   VAR
      s_UDT_MessageArray { ExternalAccessible := 'False'; ExternalVisible := 'False'; ExternalWritable := 'False'; S7_SetPoint := 'False'} : "UDT_MessageV2";   // Message array byte
      s_UDT_MessageHeader { ExternalAccessible := 'False'; ExternalVisible := 'False'; ExternalWritable := 'False'; S7_SetPoint := 'False'} : "UDT_MFCSortMessageHeader";   // Message header
      s_F_TRIG_SendAllStatuses {InstructionName := 'F_TRIG'; LibVersion := '1.0'; ExternalAccessible := 'False'; ExternalVisible := 'False'; ExternalWritable := 'False'; S7_SetPoint := 'False'} : F_TRIG;   // Falling edge trigger from signal send all statuses
      ss_MessageBody { ExternalAccessible := 'False'; ExternalVisible := 'False'; ExternalWritable := 'False'} : Struct   // Message body
         MsgID { ExternalAccessible := 'False'; ExternalVisible := 'False'; ExternalWritable := 'False'} : Word;   // Message ID
         MsgLength { ExternalAccessible := 'False'; ExternalVisible := 'False'; ExternalWritable := 'False'} : Word;   // Message length
         SystemStatus { ExternalAccessible := 'False'; ExternalVisible := 'False'; ExternalWritable := 'False'} : Byte;   // System status
         SystemMode { ExternalAccessible := 'False'; ExternalVisible := 'False'; ExternalWritable := 'False'} : Word;   // System mode
         Eom { ExternalAccessible := 'False'; ExternalVisible := 'False'; ExternalWritable := 'False'} : Byte;   // End of message
      END_STRUCT;
      ss_Status { ExternalAccessible := 'False'; ExternalVisible := 'False'; ExternalWritable := 'False'} : Struct   // Status structure
         FIFOStatus { ExternalAccessible := 'False'; ExternalVisible := 'False'; ExternalWritable := 'False'} : "UDT_FifoStatus";
         FIFOError { ExternalAccessible := 'False'; ExternalVisible := 'False'; ExternalWritable := 'False'; S7_SetPoint := 'True'} : Bool;   //  FIFO error
         FIFOWarning { ExternalAccessible := 'False'; ExternalVisible := 'False'; ExternalWritable := 'False'; S7_SetPoint := 'True'} : Bool;   // FIFO warning
         InvalidMessageArraySize { ExternalAccessible := 'False'; ExternalVisible := 'False'; ExternalWritable := 'False'} : Bool;   // Message array is too short for message
         InvalidTimeInterval { ExternalAccessible := 'False'; ExternalVisible := 'False'; ExternalWritable := 'False'} : Bool;   // Heartbeat time interval lower than zero
      END_STRUCT;
      sdi_SerializePosition { ExternalAccessible := 'False'; ExternalVisible := 'False'; ExternalWritable := 'False'} : DInt;   // Position in array where serialize finished writing data +1
      si_MaximumMessageLength { ExternalAccessible := 'False'; ExternalVisible := 'False'; ExternalWritable := 'False'} : Int;   // Maximum number of elements in message array
      si_SerializeStatus { ExternalAccessible := 'False'; ExternalVisible := 'False'; ExternalWritable := 'False'} : Int;   // Function serialize status
      si_SystemStatus { ExternalAccessible := 'False'; ExternalVisible := 'False'; ExternalWritable := 'False'} : Int := 0;   // 0 - System stopped, 1 - System running
      sw_SystemMode { ExternalAccessible := 'False'; ExternalVisible := 'False'; ExternalWritable := 'False'} : Word := 0;   // Bit value according to the documentation
      si_Old_SystemStatus { ExternalAccessible := 'False'; ExternalVisible := 'False'; ExternalWritable := 'False'} : Int := 0;   // Data from previous PLC cycle: 0 - System stopped, 1 - System running
      sw_Old_SystemMode { ExternalAccessible := 'False'; ExternalVisible := 'False'; ExternalWritable := 'False'} : Word := 0;   // Bit value according to the documentation
      sx_NewData { ExternalAccessible := 'False'; ExternalVisible := 'False'; ExternalWritable := 'False'} : Bool;   // True - send a message to the MFC
   END_VAR

   VAR CONSTANT
      ci_MessageLength : Word := 16#0006;   // 10#0006 = 16#0006 - Message length
      ci_Som : Byte := 16#FD;   // Start of message
      ci_Eom : Byte := 16#FE;   // End of message
      ci_MsgID : Word := 16#00CC;   // 10#0204 = 16#00CC - Message ID
      ci_MsgLength : Word := 16#0002;   // 10#0002 = 16#0002 - Message length
   END_VAR


BEGIN
	(*
	----------------------------------------------------------------------------------------
	|                                                                                      |
	|  Copyright  2023             FORTNA Europe BV                                        |
	|  All Rights Reserved         Netherlands                                             |
	|                                                                                      |
	----------------------------------------------------------------------------------------
	Version history:
	Date        | Version   | Author       | Remark
	----------------------------------------------------------------------------------------
	25/04/2023  | 1.0       | S. Nikodem   | Release TIA 17 | DHL Munich 2023
	13/09/2023  | 1.1       | S. Nikodem   | Change type of variable System mode to word
	20/10/2023  | 1.2       | S. Nikodem   | Added "ix_SendAllStatuses" input and update for Serialize structure
	13/03/2023  | 1.3       | S. Nieswiec  | Updated for new Baseline
	02/05/2024  | 1.4       | J.Majer      | Datatype conversions changed from automatic to explicit, to accomodate IEC 61131-3 standard

	*)

	REGION 1 – FIFO header status update

	    // Mode 'S' - FIFO register status update.
	    "FC_Fifo"(ic_Mode := 'S',
	              qUDT_Status => #ss_Status.FIFOStatus,
	              qx_Error => #ss_Status.FIFOError,
	              qx_Warning => #ss_Status.FIFOWarning,
	              iqv_Data := #s_UDT_MessageArray,
	              iqUDT_FifoHeader := #iq_UDT_FifoHeader,
	              iqv_DataBuffer := #iqa_FifoData);

	END_REGION

	REGION 2 – Data preparation

	    // Prepare trigger
	    #s_F_TRIG_SendAllStatuses(CLK := #ix_SendAllStatuses);

	    // Data preparation
	    //  1 - System stopped, 2 - System running
	    #si_SystemStatus := #ii_SystemStatus;
	    // Bit value according to the documentation
	    #sw_SystemMode := #iw_SystemMode;

	    //Check if the data from the previous PLC cycle differs, if so, send a message to the MFC.
	    #sx_NewData := (#si_Old_SystemStatus <> #si_SystemStatus) OR (#sw_Old_SystemMode <> #sw_SystemMode) OR #s_F_TRIG_SendAllStatuses.Q;

	    // Copy data
	    #si_Old_SystemStatus := #si_SystemStatus;
	    #sw_Old_SystemMode := #sw_SystemMode;

	END_REGION

	REGION 3 – Message array size validation

	    // Get size of the array.
	    #si_MaximumMessageLength := "FC_GetNrOfArrayEl"(#s_UDT_MessageArray.Bytes);

	    // Message array size validation.
	    #ss_Status.InvalidMessageArraySize := WORD_TO_INT(#ci_MessageLength) > #si_MaximumMessageLength;

	END_REGION

	REGION 4 – Message preparation

	    // FIFO full check.
	    IF NOT #iq_UDT_FifoHeader.Status.Full
	    THEN
	        // Errors and send pulse check.
	        IF NOT #ss_Status.FIFOError
	            AND NOT #ss_Status.InvalidMessageArraySize
	            AND #sx_NewData
	        THEN

	            REGION 4.1 – Header preparation

	                // Check sequence number. If it is equal or greater than 255 reset it to 1.
	                IF #iqi_MessageSequenceNumber <= 255
	                THEN
	                    #iqi_MessageSequenceNumber += 1;
	                ELSE
	                    #iqi_MessageSequenceNumber := 1;
	                END_IF;

	                // Write parts of the header into structure.
	                #s_UDT_MessageHeader.SOM := #ci_Som;
	                #s_UDT_MessageHeader.SourceNode := INT_TO_BYTE(#ii_SourceNode);
	                #s_UDT_MessageHeader.DestinationNode := INT_TO_BYTE(#ii_DestinationNode);
	                #s_UDT_MessageHeader.SeqNumber := INT_TO_BYTE(#iqi_MessageSequenceNumber);
	                #s_UDT_MessageHeader.DataLength := #ci_MessageLength;
	                #s_UDT_MessageHeader.NumMsg := 1;

	                // Write parts of the body into structure.
	                #ss_MessageBody.MsgID := #ci_MsgID;
	                #ss_MessageBody.MsgLength := #ci_MsgLength;
	                #ss_MessageBody.SystemStatus := INT_TO_BYTE(#si_SystemStatus);
	                #ss_MessageBody.SystemMode := #sw_SystemMode;
	                #ss_MessageBody.Eom := #ci_Eom;

	            END_REGION

	            REGION 4.2 – Convert message into array of bytes

	                // Initialize the header serialize position and convert header structure into array of bytes.
	                #sdi_SerializePosition := 0;
	                #si_SerializeStatus := Serialize(SRC_VARIABLE := #s_UDT_MessageHeader,
	                                                 DEST_ARRAY => #s_UDT_MessageArray.Bytes,
	                                                 POS := #sdi_SerializePosition);

	                #si_SerializeStatus := Serialize(SRC_VARIABLE := #ss_MessageBody.MsgID,
	                                                 DEST_ARRAY => #s_UDT_MessageArray.Bytes,
	                                                 POS := #sdi_SerializePosition);

	                #si_SerializeStatus := Serialize(SRC_VARIABLE := #ss_MessageBody.MsgLength,
	                                                 DEST_ARRAY => #s_UDT_MessageArray.Bytes,
	                                                 POS := #sdi_SerializePosition);

	                #si_SerializeStatus := Serialize(SRC_VARIABLE := #ss_MessageBody.SystemStatus,
	                                                 DEST_ARRAY => #s_UDT_MessageArray.Bytes,
	                                                 POS := #sdi_SerializePosition);

	                #si_SerializeStatus := Serialize(SRC_VARIABLE := #ss_MessageBody.SystemMode,
	                                                 DEST_ARRAY => #s_UDT_MessageArray.Bytes,
	                                                 POS := #sdi_SerializePosition);

	                #si_SerializeStatus := Serialize(SRC_VARIABLE := #ss_MessageBody.Eom,
	                                                 DEST_ARRAY => #s_UDT_MessageArray.Bytes,
	                                                 POS := #sdi_SerializePosition);

	            END_REGION

	            REGION 4.3 – Write message into the FIFO buffer

	                // Mode 'W' - Write FIFO record.
	                "FC_Fifo"(ic_Mode := 'W',
	                          qUDT_Status => #ss_Status.FIFOStatus,
	                          qx_Error => #ss_Status.FIFOError,
	                          qx_Warning => #ss_Status.FIFOWarning,
	                          iqv_Data := #s_UDT_MessageArray,
	                          iqUDT_FifoHeader := #iq_UDT_FifoHeader,
	                          iqv_DataBuffer := #iqa_FifoData);

	            END_REGION

	        END_IF;
	    ELSE
	        // If FIFO is full set FIFO main and FIFO full errors.
	        #ss_Status.FIFOError := TRUE;
	        #ss_Status.FIFOStatus.FifoFull := TRUE;
	    END_IF;

	END_REGION

	REGION 5 - Status

	    // Parametrization collective error output.
	    #qx_Error :=
	    #ss_Status.FIFOError
	    OR #ss_Status.InvalidTimeInterval
	    OR #ss_Status.InvalidMessageArraySize;

	    // Parametrization collective warning output.
	    #qx_Warning := #ss_Status.FIFOWarning;

	END_REGION
END_FUNCTION_BLOCK

FUNCTION_BLOCK "FB_MFC_Sort_COY_Result"
{ S7_Optimized_Access := 'TRUE' }
VERSION : 0.1
// ATTRIBUTES
// AUTO_NUMBER = True
// BLOCK_NUMBER = 117
// END_ATTRIBUTES
   VAR_INPUT
      ii_GINRangeStart { ExternalAccessible := 'False'; ExternalVisible := 'False'; ExternalWritable := 'False'} : Int := 0;   // GIN range start value
      ii_GINRangeEnd { ExternalAccessible := 'False'; ExternalVisible := 'False'; ExternalWritable := 'False'} : Int := 0;   // GIN range end value
      is_ObjectID { ExternalAccessible := 'False'; ExternalVisible := 'False'; ExternalWritable := 'False'} : String[10];   // Recived parcel identifier
      ii_SourceNode { ExternalAccessible := 'False'; ExternalVisible := 'False'; ExternalWritable := 'False'} : Int;   // ID Source Node
      ii_DestinationNode { ExternalAccessible := 'False'; ExternalVisible := 'False'; ExternalWritable := 'False'} : Int;   // ID Destination Node
   END_VAR

   VAR_OUTPUT
      qx_Error { ExternalAccessible := 'False'; ExternalVisible := 'False'; ExternalWritable := 'False'} : Bool;   // TRUE when collective block error occurred
      qx_Warning { ExternalAccessible := 'False'; ExternalVisible := 'False'; ExternalWritable := 'False'} : Bool;   // TRUE when collective block warning occurred
   END_VAR

   VAR_IN_OUT
      iq_UDT_FifoHeader : "UDT_FifoHeader";   // FIFO header
      iqa_FifoData : Array[*] of "UDT_MessageV2";   // FIFO data buffer
      iqi_MessageSequenceNumber { ExternalAccessible := 'False'; ExternalVisible := 'False'; ExternalWritable := 'False'} : Int;   // Message number
   END_VAR

   VAR
      ss_FB_HeartbeatPulse { ExternalAccessible := 'False'; ExternalVisible := 'False'; ExternalWritable := 'False'; S7_SetPoint := 'False'} : "FB_Pulse";   // Heartbeat send pulse generator
      s_UDT_MessageArray { ExternalAccessible := 'False'; ExternalVisible := 'False'; ExternalWritable := 'False'; S7_SetPoint := 'False'} : "UDT_MessageV2";   // Message array byte
      s_UDT_MessageHeader { ExternalAccessible := 'False'; ExternalVisible := 'False'; ExternalWritable := 'False'; S7_SetPoint := 'False'} : "UDT_MFCSortMessageHeader";   // Message header
      ss_MessageBody { ExternalAccessible := 'False'; ExternalVisible := 'False'; ExternalWritable := 'False'} : Struct   // Message body
         MsgID { ExternalAccessible := 'False'; ExternalVisible := 'False'; ExternalWritable := 'False'} : Word;   // Message ID
         MsgLength { ExternalAccessible := 'False'; ExternalVisible := 'False'; ExternalWritable := 'False'} : Word;   // Message length
         VID { ExternalAccessible := 'False'; ExternalVisible := 'False'; ExternalWritable := 'False'} : Array[1..16] of Byte;   // Virtual Item Identifier
         PieceID { ExternalAccessible := 'False'; ExternalVisible := 'False'; ExternalWritable := 'False'} : Array[1..40] of Byte;   // Piece ID
         Group { ExternalAccessible := 'False'; ExternalVisible := 'False'; ExternalWritable := 'False'} : Byte;   // Group
         Level { ExternalAccessible := 'False'; ExternalVisible := 'False'; ExternalWritable := 'False'} : Byte;   // Level
         Result { ExternalAccessible := 'False'; ExternalVisible := 'False'; ExternalWritable := 'False'} : Byte;   // Result
         Eom { ExternalAccessible := 'False'; ExternalVisible := 'False'; ExternalWritable := 'False'} : Byte;   // End of message
      END_STRUCT;
      ss_MessageData { ExternalAccessible := 'False'; ExternalVisible := 'False'; ExternalWritable := 'False'} : Struct   // Message data
         VID { ExternalAccessible := 'False'; ExternalVisible := 'False'; ExternalWritable := 'False'} : Array[1..16] of Byte;   // Virtual Item Identifier
         PieceID { ExternalAccessible := 'False'; ExternalVisible := 'False'; ExternalWritable := 'False'} : Array[1..40] of Byte;   // Piece ID
         Group { ExternalAccessible := 'False'; ExternalVisible := 'False'; ExternalWritable := 'False'} : String[1];   // Group
         Level { ExternalAccessible := 'False'; ExternalVisible := 'False'; ExternalWritable := 'False'} : String[1];   // Level
         Result { ExternalAccessible := 'False'; ExternalVisible := 'False'; ExternalWritable := 'False'} : String[1];   // Result
      END_STRUCT;
      ss_Status { ExternalAccessible := 'False'; ExternalVisible := 'False'; ExternalWritable := 'False'} : Struct   // Status structure
         FIFOStatus { ExternalAccessible := 'False'; ExternalVisible := 'False'; ExternalWritable := 'False'} : "UDT_FifoStatus";
         FIFOError { ExternalAccessible := 'False'; ExternalVisible := 'False'; ExternalWritable := 'False'; S7_SetPoint := 'True'} : Bool;   //  FIFO error
         FIFOWarning { ExternalAccessible := 'False'; ExternalVisible := 'False'; ExternalWritable := 'False'; S7_SetPoint := 'True'} : Bool;   // FIFO warning
         InvalidMessageArraySize { ExternalAccessible := 'False'; ExternalVisible := 'False'; ExternalWritable := 'False'} : Bool;   // Message array is too short for message
         InvalidTimeInterval { ExternalAccessible := 'False'; ExternalVisible := 'False'; ExternalWritable := 'False'} : Bool;   // Heartbeat time interval lower than zero
      END_STRUCT;
      sS_Old_Object_ID { ExternalAccessible := 'False'; ExternalVisible := 'False'; ExternalWritable := 'False'} : String[10];   // Value from previous PLC cycle
      sdi_SerializePosition { ExternalAccessible := 'False'; ExternalVisible := 'False'; ExternalWritable := 'False'} : DInt;   // Position in array where serialize finished writing data +1
      si_MaximumMessageLength { ExternalAccessible := 'False'; ExternalVisible := 'False'; ExternalWritable := 'False'} : Int;   // Maximum number of elements in message array
      si_SerializeStatus { ExternalAccessible := 'False'; ExternalVisible := 'False'; ExternalWritable := 'False'} : Int;   // Function serialize status
      sx_NewData { ExternalAccessible := 'False'; ExternalVisible := 'False'; ExternalWritable := 'False'} : Bool;   // True - send a message to the MFC
   END_VAR

   VAR_TEMP
      ti_Loop_GIN : Int;   // Loop counter for DB_GIN
      ti_Loop : Int;   // Loop counter
   END_VAR

   VAR CONSTANT
      ci_MessageLength : Word := 16#003F;   // 10#0063 = 16#003F - Message length
      ci_MsgID : Word := 16#0137;   // 10#0311 = 16#0137 - Message ID
      ci_MsgLength : Word := 16#003B;   // 10#0059 = 16#003B - Message length
      ci_Som : Byte := 16#FD;   // Start of message
      ci_Eom : Byte := 16#FE;   // End of message
   END_VAR


BEGIN
	(*
	----------------------------------------------------------------------------------------
	|                                                                                      |
	|  Copyright  2023             FORTNA Europe BV                                        |
	|  All Rights Reserved         Netherlands                                             |
	|                                                                                      |
	----------------------------------------------------------------------------------------
	Version history:
	Date        | Version   | Author       | Remark
	----------------------------------------------------------------------------------------
	24/04/2023  | 1.0       | S. Nikodem   | Release TIA 17 | DHL Munich 2023
	03/10/2023  | 1.1       | S. Nikodem   | Update
	13/03/2023  | 1.2       | S. Nieswiec  | Updated for new Baseline
	02/05/2024  | 1.3       | J.Majer      | Datatype conversions changed from automatic to explicit, to accomodate IEC 61131-3 standard
	*)

	REGION 1 – FIFO header status update

	    // Mode 'S' - FIFO register status update.
	    "FC_Fifo"(ic_Mode := 'S',
	              qUDT_Status => #ss_Status.FIFOStatus,
	              qx_Error => #ss_Status.FIFOError,
	              qx_Warning => #ss_Status.FIFOWarning,
	              iqv_Data := #s_UDT_MessageArray,
	              iqUDT_FifoHeader := #iq_UDT_FifoHeader,
	              iqv_DataBuffer := #iqa_FifoData);

	END_REGION

	REGION 2 – Data preparation

	    //Generation message when is new parcel
	    #sx_NewData := (#is_ObjectID <> #sS_Old_Object_ID) AND NOT (#is_ObjectID = '');
	    // Save last value
	    #sS_Old_Object_ID := #is_ObjectID;

	    IF #sx_NewData THEN

	        FOR #ti_Loop_GIN := #ii_GINRangeStart TO #ii_GINRangeEnd DO

	            IF "DB_GIN".GIN[#ti_Loop_GIN].DHL.ObjectID = #is_ObjectID THEN

	                //VID
	                FOR #ti_Loop := 1 TO 16 DO

	                    #ss_MessageData.VID[#ti_Loop] := CHAR_TO_BYTE("DB_GIN".GIN[#ti_Loop_GIN].DHL.VID[#ti_Loop]);

	                END_FOR;

	                //Piece ID
	                FOR #ti_Loop := 1 TO 40 DO

	                    #ss_MessageData.PieceID[#ti_Loop] := CHAR_TO_BYTE("DB_GIN".GIN[#ti_Loop_GIN].DHL.PieceID[#ti_Loop]);

	                END_FOR;

	                //Group
	                #ss_MessageData.Group := "DB_GIN".GIN[#ti_Loop_GIN].DHL.Xray.Group;

	                //Level
	                #ss_MessageData.Level := "DB_GIN".GIN[#ti_Loop_GIN].DHL.Xray.Level;

	                //Result
	                #ss_MessageData.Result := "DB_GIN".GIN[#ti_Loop_GIN].DHL.Xray.Result;

	            END_IF;

	        END_FOR;

	    END_IF;

	END_REGION

	REGION 3 – Message array size validation

	    // Get size of the array.
	    #si_MaximumMessageLength := "FC_GetNrOfArrayEl"(#s_UDT_MessageArray.Bytes);

	    // Message array size validation.
	    #ss_Status.InvalidMessageArraySize := WORD_TO_INT(#ci_MessageLength) > #si_MaximumMessageLength;

	END_REGION


	REGION 4 – Message preparation

	    // FIFO full check.
	    IF NOT #iq_UDT_FifoHeader.Status.Full
	    THEN
	        // Errors and send pulse check.
	        IF NOT #ss_Status.FIFOError
	            AND NOT #ss_Status.InvalidMessageArraySize
	            AND #sx_NewData
	        THEN

	            REGION 4.1 – Header preparation

	                // Check sequence number. If it is equal or greater than 255 reset it to 1.
	                IF #iqi_MessageSequenceNumber <= 255
	                THEN
	                    #iqi_MessageSequenceNumber += 1;
	                ELSE
	                    #iqi_MessageSequenceNumber := 1;
	                END_IF;

	                // Write parts of the header into structure.
	                #s_UDT_MessageHeader.SOM := #ci_Som;
	                #s_UDT_MessageHeader.SourceNode := INT_TO_BYTE(#ii_SourceNode);
	                #s_UDT_MessageHeader.DestinationNode := INT_TO_BYTE(#ii_DestinationNode);
	                #s_UDT_MessageHeader.SeqNumber := INT_TO_BYTE(#iqi_MessageSequenceNumber);
	                #s_UDT_MessageHeader.DataLength := #ci_MessageLength;
	                #s_UDT_MessageHeader.NumMsg := 1;

	                // Write parts of the body into structure.
	                #ss_MessageBody.MsgID := #ci_MsgID;
	                #ss_MessageBody.MsgLength := #ci_MsgLength;
	                #ss_MessageBody.VID := #ss_MessageData.VID;
	                #ss_MessageBody.PieceID := #ss_MessageData.PieceID;
	                #ss_MessageBody.Group := CHAR_TO_BYTE(STRING_TO_CHAR(#ss_MessageData.Group));
	                #ss_MessageBody.Level := CHAR_TO_BYTE(STRING_TO_CHAR(#ss_MessageData.Level));
	                #ss_MessageBody.Result := CHAR_TO_BYTE(STRING_TO_CHAR(#ss_MessageData.Result));
	                #ss_MessageBody.Eom := #ci_Eom;

	            END_REGION

	            REGION 4.2 – Convert message into array of bytes

	                // Initialize the header serialize position and convert header structure into array of bytes.
	                #sdi_SerializePosition := 0;
	                #si_SerializeStatus := Serialize(SRC_VARIABLE := #s_UDT_MessageHeader,
	                                                 DEST_ARRAY => #s_UDT_MessageArray.Bytes,
	                                                 POS := #sdi_SerializePosition);

	                // Initialize the body serialize position and convert header structure into array of bytes
	                #si_SerializeStatus := Serialize(SRC_VARIABLE := #ss_MessageBody,
	                                                 DEST_ARRAY => #s_UDT_MessageArray.Bytes,
	                                                 POS := #sdi_SerializePosition);

	            END_REGION

	            REGION 4.3 – Write message into the FIFO buffer

	                // Mode 'W' - Write FIFO record.
	                "FC_Fifo"(ic_Mode := 'W',
	                          qUDT_Status => #ss_Status.FIFOStatus,
	                          qx_Error => #ss_Status.FIFOError,
	                          qx_Warning => #ss_Status.FIFOWarning,
	                          iqv_Data := #s_UDT_MessageArray,
	                          iqUDT_FifoHeader := #iq_UDT_FifoHeader,
	                          iqv_DataBuffer := #iqa_FifoData);

	            END_REGION

	        END_IF;
	    ELSE
	        // If FIFO is full set FIFO main and FIFO full errors.
	        #ss_Status.FIFOError := TRUE;
	        #ss_Status.FIFOStatus.FifoFull := TRUE;
	    END_IF;

	END_REGION

	REGION 5 - Status

	    // Parametrization collective error output.
	    #qx_Error :=
	    #ss_Status.FIFOError
	    OR #ss_Status.InvalidTimeInterval
	    OR #ss_Status.InvalidMessageArraySize;

	    // Parametrization collective warning output.
	    #qx_Warning := #ss_Status.FIFOWarning;

	END_REGION
END_FUNCTION_BLOCK

FUNCTION_BLOCK "FB_MFC_Sort_COY_RegInfo"
{ S7_Optimized_Access := 'TRUE' }
VERSION : 0.1
// ATTRIBUTES
// AUTO_NUMBER = True
// BLOCK_NUMBER = 116
// END_ATTRIBUTES
   VAR_INPUT
      is_ObjectID { ExternalAccessible := 'False'; ExternalVisible := 'False'; ExternalWritable := 'False'} : String[10];   // Parcel identifier
      ii_XrayLocation { ExternalAccessible := 'False'; ExternalVisible := 'False'; ExternalWritable := 'False'} : Int;   // X-ray location
      ii_SourceNode { ExternalAccessible := 'False'; ExternalVisible := 'False'; ExternalWritable := 'False'} : Int;   // ID Source Node
      ii_DestinationNode { ExternalAccessible := 'False'; ExternalVisible := 'False'; ExternalWritable := 'False'} : Int;   // ID Destination Node
   END_VAR

   VAR_OUTPUT
      qx_Error { ExternalAccessible := 'False'; ExternalVisible := 'False'; ExternalWritable := 'False'} : Bool;   // TRUE when collective block error occurred
      qx_Warning { ExternalAccessible := 'False'; ExternalVisible := 'False'; ExternalWritable := 'False'} : Bool;   // TRUE when collective block warning occurred
   END_VAR

   VAR_IN_OUT
      iq_UDT_FifoHeader : "UDT_FifoHeader";   // FIFO header
      iqa_FifoData : Array[*] of "UDT_MessageV2";   // FIFO data buffer
      iqi_MessageSequenceNumber { ExternalAccessible := 'False'; ExternalVisible := 'False'; ExternalWritable := 'False'} : Int;   // Message number
   END_VAR

   VAR
      ss_FB_HeartbeatPulse { ExternalAccessible := 'False'; ExternalVisible := 'False'; ExternalWritable := 'False'; S7_SetPoint := 'False'} : "FB_Pulse";   // Heartbeat send pulse generator
      s_UDT_MessageArray { ExternalAccessible := 'False'; ExternalVisible := 'False'; ExternalWritable := 'False'; S7_SetPoint := 'False'} : "UDT_MessageV2";   // Message array byte
      s_UDT_MessageHeader { ExternalAccessible := 'False'; ExternalVisible := 'False'; ExternalWritable := 'False'; S7_SetPoint := 'False'} : "UDT_MFCSortMessageHeader";   // Message header
      ss_MessageBody { ExternalAccessible := 'False'; ExternalVisible := 'False'; ExternalWritable := 'False'} : Struct   // Message body
         MsgID { ExternalAccessible := 'False'; ExternalVisible := 'False'; ExternalWritable := 'False'} : Word;   // Message ID
         MsgLength { ExternalAccessible := 'False'; ExternalVisible := 'False'; ExternalWritable := 'False'} : Word;   // Message length
         ObjectID { ExternalAccessible := 'False'; ExternalVisible := 'False'; ExternalWritable := 'False'} : DWord;   // Parcel identifier
         XrayLocation { ExternalAccessible := 'False'; ExternalVisible := 'False'; ExternalWritable := 'False'} : Word;
         Eom { ExternalAccessible := 'False'; ExternalVisible := 'False'; ExternalWritable := 'False'} : Byte;   // End of message
      END_STRUCT;
      ss_Status { ExternalAccessible := 'False'; ExternalVisible := 'False'; ExternalWritable := 'False'} : Struct   // Status structure
         FIFOStatus { ExternalAccessible := 'False'; ExternalVisible := 'False'; ExternalWritable := 'False'} : "UDT_FifoStatus";
         FIFOError { ExternalAccessible := 'False'; ExternalVisible := 'False'; ExternalWritable := 'False'; S7_SetPoint := 'True'} : Bool;   //  FIFO error
         FIFOWarning { ExternalAccessible := 'False'; ExternalVisible := 'False'; ExternalWritable := 'False'; S7_SetPoint := 'True'} : Bool;   // FIFO warning
         InvalidMessageArraySize { ExternalAccessible := 'False'; ExternalVisible := 'False'; ExternalWritable := 'False'} : Bool;   // Message array is too short for message
         InvalidTimeInterval { ExternalAccessible := 'False'; ExternalVisible := 'False'; ExternalWritable := 'False'} : Bool;   // Heartbeat time interval lower than zero
      END_STRUCT;
      si_Old_Object_ID { ExternalAccessible := 'False'; ExternalVisible := 'False'; ExternalWritable := 'False'} : String[10];   // Value from previous PLC cycle
      sdi_SerializePosition { ExternalAccessible := 'False'; ExternalVisible := 'False'; ExternalWritable := 'False'} : DInt;   // Position in array where serialize finished writing data +1
      si_MaximumMessageLength { ExternalAccessible := 'False'; ExternalVisible := 'False'; ExternalWritable := 'False'} : Int;   // Maximum number of elements in message array
      si_SerializeStatus { ExternalAccessible := 'False'; ExternalVisible := 'False'; ExternalWritable := 'False'} : Int;   // Function serialize status
      sx_NewData { ExternalAccessible := 'False'; ExternalVisible := 'False'; ExternalWritable := 'False'} : Bool;   // True - send a message to the MFC
   END_VAR

   VAR_TEMP
      tudi_Temp : UDInt;   // temporarry variable
   END_VAR

   VAR CONSTANT
      ci_MessageLength : Word := 16#0008;   // 10#0008 = 16#0008 - Message length
      ci_MsgID : Word := 16#0136;   // 10#0310 = 16#0136 - Message ID
      ci_MsgLength : Word := 16#0004;   // 10#0004 = 16#0004 - Message length
      ci_Som : Byte := 16#FD;   // Start of message
      ci_Eom : Byte := 16#FE;   // End of message
   END_VAR


BEGIN
	(*
	----------------------------------------------------------------------------------------
	|                                                                                      |
	|  Copyright  2023             FORTNA Europe BV                                        |
	|  All Rights Reserved         Netherlands                                             |
	|                                                                                      |
	----------------------------------------------------------------------------------------
	Version history:
	Date        | Version   | Author       | Remark
	----------------------------------------------------------------------------------------
	24/05/2023  | 1.0       | S. Nikodem   | Release TIA 17 | DHL Munich 2023
	13/03/2023  | 1.1       | S. Nieswiec  | Updated for new Baseline
	*)

	REGION 1 – FIFO header status update

	    // Mode 'S' - FIFO register status update.
	    "FC_Fifo"(ic_Mode := 'S',
	              qUDT_Status => #ss_Status.FIFOStatus,
	              qx_Error => #ss_Status.FIFOError,
	              qx_Warning => #ss_Status.FIFOWarning,
	              iqv_Data := #s_UDT_MessageArray,
	              iqUDT_FifoHeader := #iq_UDT_FifoHeader,
	              iqv_DataBuffer := #iqa_FifoData);

	END_REGION

	REGION 2 – Data preparation

	    //Send message when is new parcel
	    #sx_NewData := (#is_ObjectID <> #si_Old_Object_ID) AND NOT (#is_ObjectID = '');
	    // Save last value
	    #si_Old_Object_ID := #is_ObjectID;

	END_REGION

	REGION 3 – Message array size validation

	    // Get size of the array.
	    #si_MaximumMessageLength := "FC_GetNrOfArrayEl"(#s_UDT_MessageArray.Bytes);

	    // Message array size validation.
	    #ss_Status.InvalidMessageArraySize := WORD_TO_INT(#ci_MessageLength) > #si_MaximumMessageLength;

	END_REGION


	REGION 4 – Message preparation

	    // FIFO full check.
	    IF NOT #iq_UDT_FifoHeader.Status.Full
	    THEN
	        // Errors and send pulse check.
	        IF NOT #ss_Status.FIFOError
	            AND NOT #ss_Status.InvalidMessageArraySize
	            AND #sx_NewData
	        THEN

	            REGION 4.1 – Header preparation

	                // Check sequence number. If it is equal or greater than 255 reset it to 1.
	                IF #iqi_MessageSequenceNumber <= 255
	                THEN
	                    #iqi_MessageSequenceNumber += 1;
	                ELSE
	                    #iqi_MessageSequenceNumber := 1;
	                END_IF;

	                // Write parts of the header into structure.
	                #s_UDT_MessageHeader.SOM := #ci_Som;
	                #s_UDT_MessageHeader.SourceNode := INT_TO_BYTE(#ii_SourceNode);
	                #s_UDT_MessageHeader.DestinationNode := INT_TO_BYTE(#ii_DestinationNode);
	                #s_UDT_MessageHeader.SeqNumber := INT_TO_BYTE(#iqi_MessageSequenceNumber);
	                #s_UDT_MessageHeader.DataLength := #ci_MessageLength;
	                #s_UDT_MessageHeader.NumMsg := 1;

	                //Convert string value to UDINT
	                #tudi_Temp := STRING_TO_UDINT(#is_ObjectID);

	                // Write parts of the body into structure.
	                #ss_MessageBody.MsgID := #ci_MsgID;
	                #ss_MessageBody.MsgLength := #ci_MsgLength;
	                #ss_MessageBody.ObjectID := UDINT_TO_DWORD(#tudi_Temp);
	                #ss_MessageBody.XrayLocation := INT_TO_WORD(#ii_XrayLocation);
	                #ss_MessageBody.Eom := #ci_Eom;

	            END_REGION

	            REGION 4.2 – Convert message into array of bytes

	                // Initialize the header serialize position and convert header structure into array of bytes.
	                #sdi_SerializePosition := 0;
	                #si_SerializeStatus := Serialize(SRC_VARIABLE := #s_UDT_MessageHeader,
	                                                 DEST_ARRAY => #s_UDT_MessageArray.Bytes,
	                                                 POS := #sdi_SerializePosition);

	                // Initialize the body serialize position and convert header structure into array of bytes
	                #si_SerializeStatus := Serialize(SRC_VARIABLE := #ss_MessageBody,
	                                                 DEST_ARRAY => #s_UDT_MessageArray.Bytes,
	                                                 POS := #sdi_SerializePosition);

	            END_REGION

	            REGION 4.3 – Write message into the FIFO buffer

	                // Mode 'W' - Write FIFO record.
	                "FC_Fifo"(ic_Mode := 'W',
	                          qUDT_Status => #ss_Status.FIFOStatus,
	                          qx_Error => #ss_Status.FIFOError,
	                          qx_Warning => #ss_Status.FIFOWarning,
	                          iqv_Data := #s_UDT_MessageArray,
	                          iqUDT_FifoHeader := #iq_UDT_FifoHeader,
	                          iqv_DataBuffer := #iqa_FifoData);

	            END_REGION

	        END_IF;
	    ELSE
	        // If FIFO is full set FIFO main and FIFO full errors.
	        #ss_Status.FIFOError := TRUE;
	        #ss_Status.FIFOStatus.FifoFull := TRUE;
	    END_IF;

	END_REGION

	REGION 5 - Status

	    // Parametrization collective error output.
	    #qx_Error :=
	    #ss_Status.FIFOError
	    OR #ss_Status.InvalidTimeInterval
	    OR #ss_Status.InvalidMessageArraySize;

	    // Parametrization collective warning output.
	    #qx_Warning := #ss_Status.FIFOWarning;

	END_REGION
END_FUNCTION_BLOCK

FUNCTION_BLOCK "FB_MFC_Sort_COY_ReceiveResult"
{ S7_Optimized_Access := 'TRUE' }
VERSION : 0.1
// ATTRIBUTES
// AUTO_NUMBER = True
// BLOCK_NUMBER = 115
// END_ATTRIBUTES
   VAR_INPUT
      is_VID { ExternalAccessible := 'False'; ExternalVisible := 'False'; ExternalWritable := 'False'} : String[16];   // Virtual Item Identifier (VID)
      is_PieceID { ExternalAccessible := 'False'; ExternalVisible := 'False'; ExternalWritable := 'False'} : String[40];   // Piece ID barcodes
      is_Group { ExternalAccessible := 'False'; ExternalVisible := 'False'; ExternalWritable := 'False'} : String[1];   // The group field is used to identify the group of the operator decisions came from in a
      is_Level { ExternalAccessible := 'False'; ExternalVisible := 'False'; ExternalWritable := 'False'} : String[1];   // Level field is used to identify which level the operator decision came from in a
      is_Result { ExternalAccessible := 'False'; ExternalVisible := 'False'; ExternalWritable := 'False'} : String[1];   // Results can be indicated with the following
      ii_SourceNode { ExternalAccessible := 'False'; ExternalVisible := 'False'; ExternalWritable := 'False'} : Int;   // ID Source Node
      ii_DestinationNode { ExternalAccessible := 'False'; ExternalVisible := 'False'; ExternalWritable := 'False'} : Int;   // ID Destination Node
   END_VAR

   VAR_OUTPUT
      qx_Error { ExternalAccessible := 'False'; ExternalVisible := 'False'; ExternalWritable := 'False'} : Bool;   // TRUE when collective block error occurred
      qx_Warning { ExternalAccessible := 'False'; ExternalVisible := 'False'; ExternalWritable := 'False'} : Bool;   // TRUE when collective block warning occurred
   END_VAR

   VAR_IN_OUT
      iq_UDT_FifoHeader : "UDT_FifoHeader";   // FIFO header
      iqa_FifoData : Array[*] of "UDT_MessageV2";   // FIFO data buffer
      iqi_MessageSequenceNumber { ExternalAccessible := 'False'; ExternalVisible := 'False'; ExternalWritable := 'False'} : Int;   // Message number
   END_VAR

   VAR
      ss_FB_HeartbeatPulse { ExternalAccessible := 'False'; ExternalVisible := 'False'; ExternalWritable := 'False'; S7_SetPoint := 'False'} : "FB_Pulse";   // Heartbeat send pulse generator
      s_UDT_MessageArray { ExternalAccessible := 'False'; ExternalVisible := 'False'; ExternalWritable := 'False'; S7_SetPoint := 'False'} : "UDT_MessageV2";   // Message array byte
      s_UDT_MessageHeader { ExternalAccessible := 'False'; ExternalVisible := 'False'; ExternalWritable := 'False'; S7_SetPoint := 'False'} : "UDT_MFCSortMessageHeader";   // Message header
      ss_MessageBody { ExternalAccessible := 'False'; ExternalVisible := 'False'; ExternalWritable := 'False'} : Struct   // Message body
         MsgID { ExternalAccessible := 'False'; ExternalVisible := 'False'; ExternalWritable := 'False'} : Word;   // Message ID
         MsgLength { ExternalAccessible := 'False'; ExternalVisible := 'False'; ExternalWritable := 'False'} : Word;   // Message length
         VID { ExternalAccessible := 'False'; ExternalVisible := 'False'; ExternalWritable := 'False'} : Array[1..16] of Byte;   // Virtual Item Identifier
         PieceID { ExternalAccessible := 'False'; ExternalVisible := 'False'; ExternalWritable := 'False'} : Array[1..40] of Byte;   // Piece ID
         Group { ExternalAccessible := 'False'; ExternalVisible := 'False'; ExternalWritable := 'False'} : Byte;   // Group
         Level { ExternalAccessible := 'False'; ExternalVisible := 'False'; ExternalWritable := 'False'} : Byte;   // Level
         Result { ExternalAccessible := 'False'; ExternalVisible := 'False'; ExternalWritable := 'False'} : Byte;   // Result
         Eom { ExternalAccessible := 'False'; ExternalVisible := 'False'; ExternalWritable := 'False'} : Byte;   // End of message
      END_STRUCT;
      ss_MessageData { ExternalAccessible := 'False'; ExternalVisible := 'False'; ExternalWritable := 'False'} : Struct   // Message data
         VID { ExternalAccessible := 'False'; ExternalVisible := 'False'; ExternalWritable := 'False'} : Array[1..16] of Byte;   // Virtual Item Identifier
         PieceID { ExternalAccessible := 'False'; ExternalVisible := 'False'; ExternalWritable := 'False'} : Array[1..40] of Byte;   // Piece ID
         Group { ExternalAccessible := 'False'; ExternalVisible := 'False'; ExternalWritable := 'False'} : String[1];   // Group
         Level { ExternalAccessible := 'False'; ExternalVisible := 'False'; ExternalWritable := 'False'} : String[1];   // Level
         Result { ExternalAccessible := 'False'; ExternalVisible := 'False'; ExternalWritable := 'False'} : String[1];   // Result
      END_STRUCT;
      ss_Status { ExternalAccessible := 'False'; ExternalVisible := 'False'; ExternalWritable := 'False'} : Struct   // Status structure
         FIFOStatus { ExternalAccessible := 'False'; ExternalVisible := 'False'; ExternalWritable := 'False'} : "UDT_FifoStatus";
         FIFOError { ExternalAccessible := 'False'; ExternalVisible := 'False'; ExternalWritable := 'False'; S7_SetPoint := 'True'} : Bool;   //  FIFO error
         FIFOWarning { ExternalAccessible := 'False'; ExternalVisible := 'False'; ExternalWritable := 'False'; S7_SetPoint := 'True'} : Bool;   // FIFO warning
         InvalidMessageArraySize { ExternalAccessible := 'False'; ExternalVisible := 'False'; ExternalWritable := 'False'} : Bool;   // Message array is too short for message
         InvalidTimeInterval { ExternalAccessible := 'False'; ExternalVisible := 'False'; ExternalWritable := 'False'} : Bool;   // Heartbeat time interval lower than zero
      END_STRUCT;
      sdi_SerializePosition { ExternalAccessible := 'False'; ExternalVisible := 'False'; ExternalWritable := 'False'} : DInt;   // Position in array where serialize finished writing data +1
      si_MaximumMessageLength { ExternalAccessible := 'False'; ExternalVisible := 'False'; ExternalWritable := 'False'} : Int;   // Maximum number of elements in message array
      si_SerializeStatus { ExternalAccessible := 'False'; ExternalVisible := 'False'; ExternalWritable := 'False'} : Int;   // Function serialize status
      sx_NewData { ExternalAccessible := 'False'; ExternalVisible := 'False'; ExternalWritable := 'False'} : Bool;   // New data received
      ss_PieceIDOld { ExternalAccessible := 'False'; ExternalVisible := 'False'; ExternalWritable := 'False'} : String[40];   // Piece ID barcodes old value
   END_VAR

   VAR_TEMP
      ti_Loop : Int;
   END_VAR

   VAR CONSTANT
      ci_MessageLength : Word := 16#003F;   // 10#0063 = 16#003F - Message length
      ci_MsgID : Word := 16#0137;   // 10#0311 = 16#0137 - Message ID
      ci_MsgLength : Word := 16#003B;   // 10#0059 = 16#003B - Message length
      ci_Som : Byte := 16#FD;   // Start of message
      ci_Eom : Byte := 16#FE;   // End of message
   END_VAR


BEGIN
	(*
	----------------------------------------------------------------------------------------
	|                                                                                      |
	|  Copyright  2023             FORTNA Europe BV                                        |
	|  All Rights Reserved         Netherlands                                             |
	|                                                                                      |
	----------------------------------------------------------------------------------------
	Version history:
	Date        | Version   | Author       | Remark
	----------------------------------------------------------------------------------------
	05/10/2023  | 1.0       | S. Nikodem   | Release TIA 17 | DHL Munich 2023
	13/03/2023  | 1.1       | S. Nieswiec  | Updated for new Baseline
	02/05/2024  | 1.2       | J.Majer      | Datatype conversions changed from automatic to explicit, to accomodate IEC 61131-3 standard
	*)

	REGION 1 – FIFO header status update

	    // Mode 'S' - FIFO register status update.
	    "FC_Fifo"(ic_Mode := 'S',
	              qUDT_Status => #ss_Status.FIFOStatus,
	              qx_Error => #ss_Status.FIFOError,
	              qx_Warning => #ss_Status.FIFOWarning,
	              iqv_Data := #s_UDT_MessageArray,
	              iqUDT_FifoHeader := #iq_UDT_FifoHeader,
	              iqv_DataBuffer := #iqa_FifoData);

	END_REGION

	REGION 2 – Data preparation

	    IF #is_PieceID <> #ss_PieceIDOld AND NOT (#ss_PieceIDOld = '') THEN

	        //Save
	        #ss_PieceIDOld := #is_PieceID;

	        //VID
	        FOR #ti_Loop := 1 TO 16 DO

	            #ss_MessageData.VID[#ti_Loop] := CHAR_TO_BYTE(#is_VID[#ti_Loop]);

	        END_FOR;

	        //Piece ID
	        FOR #ti_Loop := 1 TO 40 DO

	            #ss_MessageData.PieceID[#ti_Loop] := CHAR_TO_BYTE(#is_PieceID[#ti_Loop]);

	        END_FOR;

	        //Group
	        #ss_MessageData.Group := #is_Group;

	        //Level
	        #ss_MessageData.Level := #is_Level;

	        //Result
	        #ss_MessageData.Result := #is_Result;

	        //New data received
	        #sx_NewData := TRUE;

	    END_IF;


	END_REGION

	REGION 3 – Message array size validation

	    // Get size of the array.
	    #si_MaximumMessageLength := "FC_GetNrOfArrayEl"(#s_UDT_MessageArray.Bytes);

	    // Message array size validation.
	    #ss_Status.InvalidMessageArraySize := WORD_TO_INT(#ci_MessageLength) > #si_MaximumMessageLength;

	END_REGION


	REGION 4 – Message preparation

	    // FIFO full check.
	    IF NOT #iq_UDT_FifoHeader.Status.Full
	    THEN
	        // Errors and send pulse check.
	        IF NOT #ss_Status.FIFOError
	            AND NOT #ss_Status.InvalidMessageArraySize
	            AND #sx_NewData
	        THEN

	            REGION 4.1 – Header preparation

	                // Check sequence number. If it is equal or greater than 255 reset it to 1.
	                IF #iqi_MessageSequenceNumber <= 255
	                THEN
	                    #iqi_MessageSequenceNumber += 1;
	                ELSE
	                    #iqi_MessageSequenceNumber := 1;
	                END_IF;

	                // Write parts of the header into structure.
	                #s_UDT_MessageHeader.SOM := #ci_Som;
	                #s_UDT_MessageHeader.SourceNode := INT_TO_BYTE(#ii_SourceNode);
	                #s_UDT_MessageHeader.DestinationNode := INT_TO_BYTE(#ii_DestinationNode);
	                #s_UDT_MessageHeader.SeqNumber := INT_TO_BYTE(#iqi_MessageSequenceNumber);
	                #s_UDT_MessageHeader.DataLength := #ci_MessageLength;
	                #s_UDT_MessageHeader.NumMsg := 1;

	                // Write parts of the body into structure.
	                #ss_MessageBody.MsgID := #ci_MsgID;
	                #ss_MessageBody.MsgLength := #ci_MsgLength;
	                #ss_MessageBody.VID := #ss_MessageData.VID;
	                #ss_MessageBody.PieceID := #ss_MessageData.PieceID;
	                #ss_MessageBody.Group := CHAR_TO_BYTE(STRING_TO_CHAR(#ss_MessageData.Group));
	                #ss_MessageBody.Level := CHAR_TO_BYTE(STRING_TO_CHAR(#ss_MessageData.Level));
	                #ss_MessageBody.Result := CHAR_TO_BYTE(STRING_TO_CHAR(#ss_MessageData.Result));
	                #ss_MessageBody.Eom := #ci_Eom;

	            END_REGION

	            REGION 4.2 – Convert message into array of bytes

	                // Initialize the header serialize position and convert header structure into array of bytes.
	                #sdi_SerializePosition := 0;
	                #si_SerializeStatus := Serialize(SRC_VARIABLE := #s_UDT_MessageHeader,
	                                                 DEST_ARRAY => #s_UDT_MessageArray.Bytes,
	                                                 POS := #sdi_SerializePosition);

	                // Initialize the body serialize position and convert header structure into array of bytes
	                #si_SerializeStatus := Serialize(SRC_VARIABLE := #ss_MessageBody,
	                                                 DEST_ARRAY => #s_UDT_MessageArray.Bytes,
	                                                 POS := #sdi_SerializePosition);

	            END_REGION

	            REGION 4.3 – Write message into the FIFO buffer

	                // Mode 'W' - Write FIFO record.
	                "FC_Fifo"(ic_Mode := 'W',
	                          qUDT_Status => #ss_Status.FIFOStatus,
	                          qx_Error => #ss_Status.FIFOError,
	                          qx_Warning => #ss_Status.FIFOWarning,
	                          iqv_Data := #s_UDT_MessageArray,
	                          iqUDT_FifoHeader := #iq_UDT_FifoHeader,
	                          iqv_DataBuffer := #iqa_FifoData);

	            END_REGION

	            //Reset
	            #sx_NewData := False;

	        END_IF;
	    ELSE
	        // If FIFO is full set FIFO main and FIFO full errors.
	        #ss_Status.FIFOError := TRUE;
	        #ss_Status.FIFOStatus.FifoFull := TRUE;
	    END_IF;

	END_REGION

	REGION 5 - Status

	    // Parametrization collective error output.
	    #qx_Error :=
	    #ss_Status.FIFOError
	    OR #ss_Status.InvalidTimeInterval
	    OR #ss_Status.InvalidMessageArraySize;

	    // Parametrization collective warning output.
	    #qx_Warning := #ss_Status.FIFOWarning;

	END_REGION
END_FUNCTION_BLOCK

FUNCTION_BLOCK "FB_MFC_Sort_TCPIPReceive"
{ S7_Optimized_Access := 'TRUE' }
VERSION : 2.3
// ATTRIBUTES
// AUTO_NUMBER = True
// BLOCK_NUMBER = 126
// END_ATTRIBUTES
   VAR_INPUT
      i_UDT_Connection { ExternalAccessible := 'False'; ExternalVisible := 'False'; ExternalWritable := 'False'} : "UDT_Connection";   // Connection parameters
      ix_EnableReceive { ExternalAccessible := 'False'; ExternalVisible := 'False'; ExternalWritable := 'False'} : Bool;   // TRUE when receive enable
      ii_DestinationID { ExternalAccessible := 'False'; ExternalVisible := 'False'; ExternalWritable := 'False'} : Int;   // Destination node ID
      ii_SourceID { ExternalAccessible := 'False'; ExternalVisible := 'False'; ExternalWritable := 'False'} : Int;   // Source node ID
   END_VAR

   VAR_OUTPUT
      qx_Error { ExternalAccessible := 'False'; ExternalVisible := 'False'; ExternalWritable := 'False'} : Bool;   // TRUE when collective block error occurred
      qx_Warning { ExternalAccessible := 'False'; ExternalVisible := 'False'; ExternalWritable := 'False'} : Bool;   // TRUE when collective block warning occurred
   END_VAR

   VAR_IN_OUT
      iq_UDT_FifoHeader : "UDT_FifoHeader";   // Fifo header
      iqs_FifoData : Variant;   // Fifo data
      iq_UDT_Statistics : "UDT_TCPIPReceiveStatisticsV2";   // Statistic structure
   END_VAR

   VAR
      s_FB_TRCV {InstructionName := 'TRCV'; LibVersion := '4.0'; ExternalAccessible := 'False'; ExternalVisible := 'False'; ExternalWritable := 'False'; S7_SetPoint := 'False'} : TRCV;   // Siemens "TRCV" block - to receive the data from TCPIP socket
      ss_TRCV { ExternalAccessible := 'False'; ExternalVisible := 'False'; ExternalWritable := 'False'} : Struct   // TRCV block interface structure
         Enable { ExternalAccessible := 'False'; ExternalVisible := 'False'; ExternalWritable := 'False'} : Bool;   //      TRCV - Enable
         NDR { ExternalAccessible := 'False'; ExternalVisible := 'False'; ExternalWritable := 'False'} : Bool;   //      TRCV - New data available
         Busy { ExternalAccessible := 'False'; ExternalVisible := 'False'; ExternalWritable := 'False'} : Bool;   //      TRCV - Busy
         Error { ExternalAccessible := 'False'; ExternalVisible := 'False'; ExternalWritable := 'False'} : Bool;   //      TRCV - Error
         Status { ExternalAccessible := 'False'; ExternalVisible := 'False'; ExternalWritable := 'False'} : Word;   //      TRCV - Status
         ReceivedLength { ExternalAccessible := 'False'; ExternalVisible := 'False'; ExternalWritable := 'False'} : UDInt;   //      TRCV - Received length
         Data { ExternalAccessible := 'False'; ExternalVisible := 'False'; ExternalWritable := 'False'} : Array[0..120] of Byte;   //      TRCV - Data
      END_STRUCT;
      ss_TRCV_empty { ExternalAccessible := 'False'; ExternalVisible := 'False'; ExternalWritable := 'False'} : Struct   // TRCV block interface structure
         Enable { ExternalAccessible := 'False'; ExternalVisible := 'False'; ExternalWritable := 'False'} : Bool;   //      TRCV - Enable
         NDR { ExternalAccessible := 'False'; ExternalVisible := 'False'; ExternalWritable := 'False'} : Bool;   //      TRCV - New data available
         Busy { ExternalAccessible := 'False'; ExternalVisible := 'False'; ExternalWritable := 'False'} : Bool;   //      TRCV - Busy
         Error { ExternalAccessible := 'False'; ExternalVisible := 'False'; ExternalWritable := 'False'} : Bool;   //      TRCV - Error
         Status { ExternalAccessible := 'False'; ExternalVisible := 'False'; ExternalWritable := 'False'} : Word;   //      TRCV - Status
         ReceivedLength { ExternalAccessible := 'False'; ExternalVisible := 'False'; ExternalWritable := 'False'} : UDInt;   //      TRCV - Received length
         Data { ExternalAccessible := 'False'; ExternalVisible := 'False'; ExternalWritable := 'False'} : Array[0..120] of Byte;   //      TRCV - Data
      END_STRUCT;
      s_UDT_MessageArray { ExternalAccessible := 'False'; ExternalVisible := 'False'; ExternalWritable := 'False'; S7_SetPoint := 'False'} : "UDT_MessageV2";   // Message byte array
   END_VAR
   VAR RETAIN
      sa_Invalid_Messages { ExternalAccessible := 'False'; ExternalVisible := 'False'; ExternalWritable := 'False'} : Array[0..99] of Struct
         Data { ExternalAccessible := 'False'; ExternalVisible := 'False'; ExternalWritable := 'False'} : Array[0..120] of Byte;
      END_STRUCT;
   END_VAR
   VAR
      ss_Status { ExternalAccessible := 'False'; ExternalVisible := 'False'; ExternalWritable := 'False'} : Struct   // Status structure
         ErrorCode { ExternalAccessible := 'False'; ExternalVisible := 'False'; ExternalWritable := 'False'} : Struct   //     Error code structure
            TRCV { ExternalAccessible := 'False'; ExternalVisible := 'False'; ExternalWritable := 'False'} : Word;   //     Siemens TRCV error code - Check documentation
         END_STRUCT;
         FIFOReceiveStatus { ExternalAccessible := 'False'; ExternalVisible := 'False'; ExternalWritable := 'False'} : "UDT_FifoStatus";   //     Receive FIFO status structure
         FIFOReceiveError { ExternalAccessible := 'False'; ExternalVisible := 'False'; ExternalWritable := 'False'; S7_SetPoint := 'True'} : Bool;   //     Receive FIFO error
         FIFOReceiveWarning { ExternalAccessible := 'False'; ExternalVisible := 'False'; ExternalWritable := 'False'; S7_SetPoint := 'True'} : Bool;   //     Receive  FIFO warning
         ReceiveError { ExternalAccessible := 'False'; ExternalVisible := 'False'; ExternalWritable := 'False'} : Bool;   //     TRCV block operation error - Check TRCVStatus
         sa_InvalidMessages { ExternalAccessible := 'False'; ExternalVisible := 'False'; ExternalWritable := 'False'} : Array[0..99] of Struct   // Invalid messages
            Data { ExternalAccessible := 'False'; ExternalVisible := 'False'; ExternalWritable := 'False'} : Array[0..120] of Byte;
         END_STRUCT;
         sui_ReceivedMessageLength { ExternalAccessible := 'False'; ExternalVisible := 'False'; ExternalWritable := 'False'} : UInt;   // Received message length
      END_STRUCT;
      sui_NumberOfReceivedMessages { ExternalAccessible := 'False'; ExternalVisible := 'False'; ExternalWritable := 'False'} : UInt;   // Number of received messages in one frame
      sdi_SerializePosition { ExternalAccessible := 'False'; ExternalVisible := 'False'; ExternalWritable := 'False'} : DInt;   // Position in array where serialize finished writing data +1
      si_MaximumMessageLength { ExternalAccessible := 'False'; ExternalVisible := 'False'; ExternalWritable := 'False'} : Int;   // Maximum message length
      si_SerializeStatus { ExternalAccessible := 'False'; ExternalVisible := 'False'; ExternalWritable := 'False'} : Int;   // Function serialize status
      si_TelegramLength { ExternalAccessible := 'False'; ExternalVisible := 'False'; ExternalWritable := 'False'} : Int;   // Telegram length - envelope + data + tail
      si_MessagesNumber { ExternalAccessible := 'False'; ExternalVisible := 'False'; ExternalWritable := 'False'} : Int;   // Messages number in Telegram
      si_Offset { ExternalAccessible := 'False'; ExternalVisible := 'False'; ExternalWritable := 'False'} : Int;   // Data offset
      si_MessageLength { ExternalAccessible := 'False'; ExternalVisible := 'False'; ExternalWritable := 'False'} : Int;   // Message length
      si_InvalidMessages { ExternalAccessible := 'False'; ExternalVisible := 'False'; ExternalWritable := 'False'} : Int;   // Arry counter invalid messages
      sx_ValidMessage { ExternalAccessible := 'False'; ExternalVisible := 'False'; ExternalWritable := 'False'} : Bool;   // Valid message signal
      sx_Watchdog { ExternalAccessible := 'False'; ExternalVisible := 'False'; ExternalWritable := 'False'} : Bool;   // Watch dog
   END_VAR

   VAR_TEMP
      ta_MessageData : Array[0..1] of Byte;   // Array of bytes
      ti_LC_TelegamBytes : Int;   // Telegram bytes loop counter
      ti_Loop_MessageCounter : Int;   // Loop counter
      ti_Loop_MessageLength : Int;   // Loop counter
   END_VAR

   VAR CONSTANT
      cc_NULL : Byte := 16#00;   // Null sign
      cb_SOM : Byte := 16#FD;   // First termination sign
      cb_EOM : Byte := 16#FE;   // Last termination sign
      ci_HeaderLength : Int := 8;   // Message header length
      ci_BodyLengthPosition : Int := 4;   // Position in header where message body length value starts
      ci_DestinationIDPosition : Int := 2;   // Position in header where destination ID
      ci_SourceIDPosition : Int := 1;   // Position in header where source ID
   END_VAR


BEGIN
	(*
	----------------------------------------------------------------------------------------
	|                                                                                      |
	|  Copyright  2023             FORTNA Europe BV                                        |
	|  All Rights Reserved         Netherlands                                             |
	|                                                                                      |
	----------------------------------------------------------------------------------------
	Version history:
	Date        | Version   | Author       | Remark
	----------------------------------------------------------------------------------------
	18/01/2023  | 1.0       | S. Nikodem   | Release TIA 17                 | DHL Munich 2023
	31/08/2023  | 2.0       | M.Diebel     | Added security to check message size
	18/12/2023  | 2.1       | S. Nikodem   | On-site update
	18/12/2023  | 2.2       | S. Nikodem   | Watchdog
	19/12/2023  | 2.3       | S. Nikodem   |
	13/03/2023  | 2.4       | S. Nieswiec  | Updated for new Baseline
	02/05/2024  | 2.5       | J.Majer      | Datatype conversions changed from automatic to explicit, to accomodate IEC 61131-3 standard

	*)

	REGION 1 – Update FIFO header status bits

	    // Mode 'S' - FIFO register status update.
	    "FC_Fifo"(ic_Mode := 'S',
	              qUDT_Status => #ss_Status.FIFOReceiveStatus,
	              qx_Error => #ss_Status.FIFOReceiveError,
	              qx_Warning => #ss_Status.FIFOReceiveWarning,
	              iqv_Data := #s_UDT_MessageArray,
	              iqUDT_FifoHeader := #iq_UDT_FifoHeader,
	              iqv_DataBuffer := #iqs_FifoData);

	END_REGION

	REGION 2 – Maximum number of message arrays elements

	    #si_MaximumMessageLength := "FC_GetNrOfArrayEl"(iv_Array := #s_UDT_MessageArray.Bytes);

	END_REGION

	REGION 3 – Receive enable

	    // Allow receiving if the connection is established and there are no FIFO errors.
	    #ss_TRCV.Enable :=
	    #ix_EnableReceive
	    AND NOT #ss_Status.FIFOReceiveError;

	END_REGION

	REGION 4 – Receive data

	    //Reset old data
	    #ss_TRCV.Data := #ss_TRCV_empty.Data;
	    #sx_ValidMessage := False;
	    #sx_Watchdog := False;

	    // Data received in an ADHOC mode - data available immediately.
	    #s_FB_TRCV(EN_R := #ss_TRCV.Enable,
	               ID := #i_UDT_Connection.ID,
	               LEN := 0,
	               ADHOC := TRUE,
	               NDR => #ss_TRCV.NDR,
	               BUSY => #ss_TRCV.Busy,
	               ERROR => #ss_TRCV.Error,
	               STATUS => #ss_TRCV.Status,
	               RCVD_LEN => #ss_TRCV.ReceivedLength,
	               DATA := #ss_TRCV.Data);

	END_REGION

	REGION 5 – Received data handling

	    // Receiving data was successful.
	    IF #ss_TRCV.NDR
	        AND NOT #ss_TRCV.Busy
	        AND NOT #ss_TRCV.Error
	        AND #ss_TRCV.ReceivedLength > 0
	    THEN

	        REGION 5.1 – Telegram handling

	            FOR #ti_LC_TelegamBytes := 0 TO (UDINT_TO_INT(#ss_TRCV.ReceivedLength) - 1) DO

	                // First termination sign found.
	                IF (#ss_TRCV.Data[#ti_LC_TelegamBytes] = #cb_SOM)
	                    AND ((#ti_LC_TelegamBytes + #ci_BodyLengthPosition + 1) <= "FC_GetNrOfArrayEl"(#ss_TRCV.Data))
	                THEN

	                    // Get the length of the telegram by extracting the body length from the telegram header.
	                    #ta_MessageData[0] := #ss_TRCV.Data[#ti_LC_TelegamBytes + #ci_BodyLengthPosition];
	                    #ta_MessageData[1] := #ss_TRCV.Data[#ti_LC_TelegamBytes + #ci_BodyLengthPosition + 1];

	                    #sdi_SerializePosition := 0;
	                    #si_SerializeStatus := Deserialize(SRC_ARRAY := #ta_MessageData,
	                                                       DEST_VARIABLE => #si_TelegramLength,
	                                                       POS := #sdi_SerializePosition);

	                    //Check if telegram lenght is correct
	                    IF #ti_LC_TelegamBytes + #si_TelegramLength + #ci_HeaderLength < "FC_GetNrOfArrayEl"(#ss_TRCV.Data) THEN

	                        //Check if on the end of the telegram is the end sign
	                        ////Watch dog
	                        IF (#ss_TRCV.Data[#ti_LC_TelegamBytes + #ci_HeaderLength] = #cb_EOM)
	                            AND (#si_TelegramLength = 0)
	                        THEN

	                            // Get the number of the messages from the telegram header.
	                            #ta_MessageData[0] := #ss_TRCV.Data[#ti_LC_TelegamBytes + #ci_BodyLengthPosition + 2];
	                            #ta_MessageData[1] := #ss_TRCV.Data[#ti_LC_TelegamBytes + #ci_BodyLengthPosition + 3];

	                            #sdi_SerializePosition := 0;
	                            #si_SerializeStatus := Deserialize(SRC_ARRAY := #ta_MessageData,
	                                                               DEST_VARIABLE => #si_MessagesNumber,
	                                                               POS := #sdi_SerializePosition);

	                            IF #si_MessagesNumber = 0 THEN

	                                #sx_Watchdog := True;
	                                #sx_ValidMessage := TRUE;

	                            END_IF;

	                        ELSIF
	                            (#ss_TRCV.Data[#ti_LC_TelegamBytes + #si_TelegramLength + #ci_HeaderLength] = #cb_EOM) THEN

	                            //Check IF the source AND destination node ID are correct
	                            IF (BYTE_TO_INT(#ss_TRCV.Data[#ti_LC_TelegamBytes + #ci_SourceIDPosition]) = #ii_SourceID)
	                                AND (BYTE_TO_INT(#ss_TRCV.Data[#ti_LC_TelegamBytes + #ci_DestinationIDPosition]) = #ii_DestinationID)
	                            THEN

	                                // Get the number of the messages from the telegram header.
	                                #ta_MessageData[0] := #ss_TRCV.Data[#ti_LC_TelegamBytes + #ci_BodyLengthPosition + 2];
	                                #ta_MessageData[1] := #ss_TRCV.Data[#ti_LC_TelegamBytes + #ci_BodyLengthPosition + 3];

	                                #sdi_SerializePosition := 0;
	                                #si_SerializeStatus := Deserialize(SRC_ARRAY := #ta_MessageData,
	                                                                   DEST_VARIABLE => #si_MessagesNumber,
	                                                                   POS := #sdi_SerializePosition);

	                                IF (#si_MessagesNumber > 0) AND (#si_MessagesNumber < 100) THEN

	                                    //Initial value
	                                    //Telegram offset
	                                    #si_Offset := #ci_HeaderLength + #ti_LC_TelegamBytes;

	                                    REGION 5.2 – Messages handling

	                                        FOR #ti_Loop_MessageCounter := 1 TO #si_MessagesNumber DO

	                                            IF (#si_Offset + 3) < "FC_GetNrOfArrayEl"(#ss_TRCV.Data) THEN

	                                                //Copy ID - word
	                                                #s_UDT_MessageArray.Bytes[0] := #ss_TRCV.Data[#si_Offset];
	                                                #s_UDT_MessageArray.Bytes[1] := #ss_TRCV.Data[#si_Offset + 1];

	                                                // Copy data length - word
	                                                #s_UDT_MessageArray.Bytes[2] := #ss_TRCV.Data[#si_Offset + 2];
	                                                #s_UDT_MessageArray.Bytes[3] := #ss_TRCV.Data[#si_Offset + 3];

	                                                #ta_MessageData[0] := #ss_TRCV.Data[#si_Offset + 2];
	                                                #ta_MessageData[1] := #ss_TRCV.Data[#si_Offset + 3];

	                                                #sdi_SerializePosition := 0;
	                                                #si_SerializeStatus := Deserialize(SRC_ARRAY := #ta_MessageData,
	                                                                                   DEST_VARIABLE => #si_MessageLength,
	                                                                                   POS := #sdi_SerializePosition);

	                                                //Copy data - byte
	                                                IF #si_MessageLength > 0 THEN

	                                                    FOR #ti_Loop_MessageLength := 0 TO #si_MessageLength DO

	                                                        #s_UDT_MessageArray.Bytes[4 + #ti_Loop_MessageLength] := #ss_TRCV.Data[#si_Offset + 4 + #ti_Loop_MessageLength];

	                                                    END_FOR;
	                                                    //Save last sign positions from message
	                                                    #si_Offset := #si_Offset + 4 + #si_MessageLength;

	                                                ELSIF #si_MessageLength = 0 THEN

	                                                    #si_Offset := #si_Offset + 4;

	                                                END_IF;

	                                                //Write message to Fifo memory
	                                                // Mode 'W' - Write FIFO record.
	                                                "FC_Fifo"(ic_Mode := 'W',
	                                                          qUDT_Status => #ss_Status.FIFOReceiveStatus,
	                                                          qx_Error => #ss_Status.FIFOReceiveError,
	                                                          qx_Warning => #ss_Status.FIFOReceiveWarning,
	                                                          iqv_Data := #s_UDT_MessageArray,
	                                                          iqUDT_FifoHeader := #iq_UDT_FifoHeader,
	                                                          iqv_DataBuffer := #iqs_FifoData);

	                                            ELSE
	                                                #iq_UDT_Statistics.InvalidMsgLength += 1;
	                                            END_IF;

	                                        END_FOR;

	                                        //Set varaible valid message
	                                        #sx_ValidMessage := True;

	                                        //Exit loop
	                                        EXIT;

	                                    END_REGION

	                                ELSE

	                                    #iq_UDT_Statistics.InvalidMsgNumber += 1;
	                                END_IF;
	                            ELSE
	                                #iq_UDT_Statistics.InvalidID += 1;
	                            END_IF;

	                        ELSE
	                            #iq_UDT_Statistics.InvalidEndSign += 1;
	                        END_IF;
	                    ELSE
	                        #iq_UDT_Statistics.InvalidTelegramLength += 1;
	                    END_IF;
	                END_IF;
	            END_FOR;

	            //Copy invalide meessage to base
	            IF NOT #sx_ValidMessage THEN

	                #iq_UDT_Statistics.InvalidMsg += 1;

	                IF #si_InvalidMessages > 99 THEN
	                    #si_InvalidMessages := 0;
	                END_IF;

	                //Save invalid data
	                #sa_Invalid_Messages[#si_InvalidMessages].Data := #ss_TRCV.Data;
	                #si_InvalidMessages += 1;

	            END_IF;

	        END_REGION

	    END_IF;

	END_REGION

	REGION 6 – Status

	    REGION 6.1 - Block status

	        // Receive error.
	        #ss_Status.ReceiveError := #ss_TRCV.Error;

	        // Parametrization collective error output.
	        #qx_Error :=
	        #ss_Status.FIFOReceiveError
	        OR #ss_Status.ReceiveError;

	        // Parametrization collective warning output.
	        #qx_Warning := #ss_Status.FIFOReceiveWarning;

	    END_REGION

	    REGION 6.2 - Error code preparation

	        IF (#ss_TRCV.#Status > 16#8000)
	            OR (#ss_TRCV.#Status = 16#0)
	        THEN
	            #ss_Status.ErrorCode.TRCV := #ss_TRCV.#Status;
	        END_IF;

	    END_REGION

	END_REGION
END_FUNCTION_BLOCK

FUNCTION_BLOCK "FB_MFC_Sort_MaintenanceCounters"
{ S7_Optimized_Access := 'TRUE' }
VERSION : 0.1
// ATTRIBUTES
// AUTO_NUMBER = True
// BLOCK_NUMBER = 121
// END_ATTRIBUTES
   VAR_INPUT
      ilr_PeriodConfig { ExternalAccessible := 'False'; ExternalVisible := 'False'; ExternalWritable := 'False'} : LReal;   // Configuration of the period how often the message should be sent [sec]
      i_UDT_ConveyorInterface { ExternalAccessible := 'False'; ExternalVisible := 'False'; ExternalWritable := 'False'} : "UDT_ConveyorInterface";   // Input conveyor interface structrue
      i_UDT_EquipmentNumber { ExternalAccessible := 'False'; ExternalVisible := 'False'; ExternalWritable := 'False'} : "UDT_EquipmentNumber";   // Item number
      ii_SourceNode { ExternalAccessible := 'False'; ExternalVisible := 'False'; ExternalWritable := 'False'} : Int;   // ID Source Node
      ii_DestinationNode { ExternalAccessible := 'False'; ExternalVisible := 'False'; ExternalWritable := 'False'} : Int;   // ID Destination Node
   END_VAR

   VAR_OUTPUT
      qx_Error { ExternalAccessible := 'False'; ExternalVisible := 'False'; ExternalWritable := 'False'} : Bool;   // TRUE when collective block error occurred
      qx_Warning { ExternalAccessible := 'False'; ExternalVisible := 'False'; ExternalWritable := 'False'} : Bool;   // TRUE when collective block warning occurred
   END_VAR

   VAR_IN_OUT
      iq_UDT_FifoHeader : "UDT_FifoHeader";   // FIFO header
      iqs_FifoData : Array[*] of "UDT_MessageV2";   // FIFO data buffer
      iqdi_MessageSequenceNumber { ExternalAccessible := 'False'; ExternalVisible := 'False'; ExternalWritable := 'False'} : Int;   // Message number
   END_VAR

   VAR
      s_UDT_MessageArray { ExternalAccessible := 'False'; ExternalVisible := 'False'; ExternalWritable := 'False'; S7_SetPoint := 'False'} : "UDT_MessageV2";   // Message array byte
      s_UDT_MessageHeader { ExternalAccessible := 'False'; ExternalVisible := 'False'; ExternalWritable := 'False'; S7_SetPoint := 'False'} : "UDT_MFCSortMessageHeader";   // Message header
      ss_MessageBody { ExternalAccessible := 'False'; ExternalVisible := 'False'; ExternalWritable := 'False'} : Struct   // Message body
         MsgID { ExternalAccessible := 'False'; ExternalVisible := 'False'; ExternalWritable := 'False'} : Word;   // Message ID
         MsgLength { ExternalAccessible := 'False'; ExternalVisible := 'False'; ExternalWritable := 'False'} : Word;   // Message length
         Group { ExternalAccessible := 'False'; ExternalVisible := 'False'; ExternalWritable := 'False'} : Word;   // Group part of item location
         Node { ExternalAccessible := 'False'; ExternalVisible := 'False'; ExternalWritable := 'False'} : Word;   // Node part of item location
         RunningTime { ExternalAccessible := 'False'; ExternalVisible := 'False'; ExternalWritable := 'False'} : DWord;   // Motor running time in seconds
         DistanceTravelled { ExternalAccessible := 'False'; ExternalVisible := 'False'; ExternalWritable := 'False'} : DWord;   // Conveyor distance travelled in mm
         "Start-Stop" { ExternalAccessible := 'False'; ExternalVisible := 'False'; ExternalWritable := 'False'} : DWord;   // Amount of start / stop actions
         Eom { ExternalAccessible := 'False'; ExternalVisible := 'False'; ExternalWritable := 'False'} : Byte;   // End of message
      END_STRUCT;
      ss_Status { ExternalAccessible := 'False'; ExternalVisible := 'False'; ExternalWritable := 'False'} : Struct   // Status structure
         FIFOStatus { ExternalAccessible := 'False'; ExternalVisible := 'False'; ExternalWritable := 'False'} : "UDT_FifoStatus";
         FIFOError { ExternalAccessible := 'False'; ExternalVisible := 'False'; ExternalWritable := 'False'; S7_SetPoint := 'True'} : Bool;   //  FIFO error
         FIFOWarning { ExternalAccessible := 'False'; ExternalVisible := 'False'; ExternalWritable := 'False'; S7_SetPoint := 'True'} : Bool;   // FIFO warning
         InvalidMessageArraySize { ExternalAccessible := 'False'; ExternalVisible := 'False'; ExternalWritable := 'False'} : Bool;   // Message array is too short for message
         InvalidTimeInterval { ExternalAccessible := 'False'; ExternalVisible := 'False'; ExternalWritable := 'False'} : Bool;   // Heartbeat time interval lower than zero
      END_STRUCT;
      s_F_TRIG_ConveyorStop {InstructionName := 'F_TRIG'; LibVersion := '1.0'; ExternalAccessible := 'False'; ExternalVisible := 'False'; ExternalWritable := 'False'; S7_SetPoint := 'False'} : F_TRIG;   // Falling edge trigger Conveyor stop
      s_R_TRIG_ConveyorStart {InstructionName := 'R_TRIG'; LibVersion := '1.0'; ExternalAccessible := 'False'; ExternalVisible := 'False'; ExternalWritable := 'False'; S7_SetPoint := 'False'} : R_TRIG;   // Rising edge trigger Conveyor start
      sdi_SerializePosition { ExternalAccessible := 'False'; ExternalVisible := 'False'; ExternalWritable := 'False'} : DInt;   // Position in array where serialize finished writing data +1
      si_MaximumMessageLength { ExternalAccessible := 'False'; ExternalVisible := 'False'; ExternalWritable := 'False'} : Int;   // Maximum number of elements in message array
      si_SerializeStatus { ExternalAccessible := 'False'; ExternalVisible := 'False'; ExternalWritable := 'False'} : Int;   // Function serialize status
      slr_RunningTimeMS { ExternalAccessible := 'False'; ExternalVisible := 'False'; ExternalWritable := 'False'} : LReal;   // Conveyor running time [ms]
      sdi_DistanceTraveled { ExternalAccessible := 'False'; ExternalVisible := 'False'; ExternalWritable := 'False'} : DInt;   // Distance traveled by conveyor
      sdi_StartStop { ExternalAccessible := 'False'; ExternalVisible := 'False'; ExternalWritable := 'False'} : DInt;   // Value of change conveyor state from start to stop and from stop to start
      sdi_RunningTime { ExternalAccessible := 'False'; ExternalVisible := 'False'; ExternalWritable := 'False'} : DInt;   // Conveyor running time [s]
      slr_PeriodMS { ExternalAccessible := 'False'; ExternalVisible := 'False'; ExternalWritable := 'False'} : LReal;   // Period to send message [ms]
      sx_SendMessage { ExternalAccessible := 'False'; ExternalVisible := 'False'; ExternalWritable := 'False'} : Bool;   // Send message to MFC
   END_VAR

   VAR CONSTANT
      ci_MessageLength : Word := 16#0014;   // 10#0020 = 16#0014 - Message length
      ci_Som : Byte := 16#FD;   // Start of message
      ci_Eom : Byte := 16#FE;   // End of message
      ci_MsgID : Word := 16#00CE;   // 10#0206 = 16#00CE - Message ID
      ci_MsgLength : Word := 16#0010;   // 10#0016 = 16#0010 - Message length
   END_VAR


BEGIN
	(*
	----------------------------------------------------------------------------------------
	|                                                                                      |
	|  Copyright  2023             FORTNA Europe BV                                        |
	|  All Rights Reserved         Netherlands                                             |
	|                                                                                      |
	----------------------------------------------------------------------------------------
	Version history:
	Date        | Version   | Author       | Remark
	----------------------------------------------------------------------------------------
	05/01/2023  | 1.0       | S. Nikodem   | Release TIA 17 | DHL Munich 2023
	09/01/2023  | 1.1       | M. Diebel    | Release TIA 17 | Convert sek from input on ms
	26/02/2024  | 1.2       | M. Diebel    | Release TIA 17 | Calculate absolute displacement
	13/03/2023  | 1.3       | S. Nieswiec  | Updated for new Baseline
	02/05/2024  | 1.4       | J.Majer      | Datatype conversions changed from automatic to explicit, to accomodate IEC 61131-3 standard

	*)

	REGION 1 – FIFO header status update

	    // Mode 'S' - FIFO register status update.
	    "FC_Fifo"(ic_Mode := 'S',
	              qUDT_Status => #ss_Status.FIFOStatus,
	              qx_Error => #ss_Status.FIFOError,
	              qx_Warning => #ss_Status.FIFOWarning,
	              iqv_Data := #s_UDT_MessageArray,
	              iqUDT_FifoHeader := #iq_UDT_FifoHeader,
	              iqv_DataBuffer := #iqs_FifoData);

	END_REGION

	REGION 2 – Data preparation

	    // Maintenance counter message is used to inform the MFC about one of three values. When one of them exceed the configured one, message is prepared and sent.
	    // Values which program is counting :
	    // - distance traveled by conveyor,
	    // - change the state of the conveyor ( stop --> start and start --> stop)
	    // - running time of the conveyor.

	    // Calculate conveyor traveled distance.
	    #sdi_DistanceTraveled += ABS(#i_UDT_ConveyorInterface.Displacement) * 10;

	    // Calculate start-stop.
	    #s_R_TRIG_ConveyorStart(CLK := #i_UDT_ConveyorInterface.RunFwd OR #i_UDT_ConveyorInterface.RunRvs);
	    #s_F_TRIG_ConveyorStop(CLK := #i_UDT_ConveyorInterface.RunRvs OR #i_UDT_ConveyorInterface.RunFwd);

	    // Increment counter on the change of the conveyor's state.
	    IF #s_R_TRIG_ConveyorStart.Q
	        OR #s_F_TRIG_ConveyorStop.Q
	    THEN
	        #sdi_StartStop += 1;
	    END_IF;

	    // Calculate running time.
	    IF #i_UDT_ConveyorInterface.RunFwd
	        OR #i_UDT_ConveyorInterface.RunRvs
	    THEN
	        #slr_RunningTimeMS += "DB_Memory".PrevCycleTime;

	        IF #slr_RunningTimeMS >= 1000
	        THEN
	            #sdi_RunningTime += 1;
	            #slr_RunningTimeMS -= 1000;
	        END_IF;

	    END_IF;

	    //Period timer
	    #slr_PeriodMS += "DB_Memory".PrevCycleTime;

	    #sx_SendMessage := #ilr_PeriodConfig * 1000.0 < #slr_PeriodMS;  //Convert sek from input on ms and compare to period

	END_REGION

	REGION 3 – Message array size validation

	    // Get size of the array.
	    #si_MaximumMessageLength := "FC_GetNrOfArrayEl"(#s_UDT_MessageArray.Bytes);

	    // Message array size validation.
	    #ss_Status.InvalidMessageArraySize := WORD_TO_INT(#ci_MessageLength) > #si_MaximumMessageLength;

	END_REGION


	REGION 4 – Message preparation

	    // FIFO full check.
	    IF NOT #iq_UDT_FifoHeader.Status.Full
	    THEN
	        // Errors and send pulse check.
	        IF NOT #ss_Status.FIFOError
	            AND NOT #ss_Status.InvalidMessageArraySize
	            AND #sx_SendMessage
	        THEN

	            //Reset counter


	            REGION 4.1 – Header preparation

	                // Check sequence number. If it is equal or greater than 255 reset it to 1.
	                IF #iqdi_MessageSequenceNumber <= 255
	                THEN
	                    #iqdi_MessageSequenceNumber += 1;
	                ELSE
	                    #iqdi_MessageSequenceNumber := 1;
	                END_IF;

	                // Write parts of the header into structure.
	                #s_UDT_MessageHeader.SOM := #ci_Som;
	                #s_UDT_MessageHeader.SourceNode := INT_TO_BYTE(#ii_SourceNode);
	                #s_UDT_MessageHeader.DestinationNode := INT_TO_BYTE(#ii_DestinationNode);
	                #s_UDT_MessageHeader.SeqNumber := INT_TO_BYTE(#iqdi_MessageSequenceNumber);
	                #s_UDT_MessageHeader.DataLength := #ci_MessageLength;
	                #s_UDT_MessageHeader.NumMsg := 1;

	                // Write parts of the body into structure.
	                #ss_MessageBody.MsgID := #ci_MsgID;
	                #ss_MessageBody.MsgLength := #ci_MsgLength;
	                #ss_MessageBody.Group := INT_TO_WORD(#i_UDT_EquipmentNumber.Group);
	                #ss_MessageBody.Node := INT_TO_WORD(#i_UDT_EquipmentNumber.Node);
	                #ss_MessageBody.RunningTime := DINT_TO_WORD(#sdi_RunningTime);
	                #ss_MessageBody.DistanceTravelled := DINT_TO_WORD(#sdi_DistanceTraveled);
	                #ss_MessageBody."Start-Stop" := DINT_TO_WORD(#sdi_StartStop);
	                #ss_MessageBody.Eom := #ci_Eom;

	            END_REGION

	            REGION 4.2 – Convert message into array of bytes

	                // Initialize the header serialize position and convert header structure into array of bytes.
	                #sdi_SerializePosition := 0;
	                #si_SerializeStatus := Serialize(SRC_VARIABLE := #s_UDT_MessageHeader,
	                                                 DEST_ARRAY => #s_UDT_MessageArray.Bytes,
	                                                 POS := #sdi_SerializePosition);

	                // Initialize the body serialize position and convert header structure into array of bytes
	                #si_SerializeStatus := Serialize(SRC_VARIABLE := #ss_MessageBody,
	                                                 DEST_ARRAY => #s_UDT_MessageArray.Bytes,
	                                                 POS := #sdi_SerializePosition);

	            END_REGION

	            REGION 4.3 – Write message into the FIFO buffer

	                // Mode 'W' - Write FIFO record.
	                "FC_Fifo"(ic_Mode := 'W',
	                          qUDT_Status => #ss_Status.FIFOStatus,
	                          qx_Error => #ss_Status.FIFOError,
	                          qx_Warning => #ss_Status.FIFOWarning,
	                          iqv_Data := #s_UDT_MessageArray,
	                          iqUDT_FifoHeader := #iq_UDT_FifoHeader,
	                          iqv_DataBuffer := #iqs_FifoData);

	            END_REGION

	            //Reset data
	            #sdi_DistanceTraveled := 0;
	            #sdi_StartStop := 0;
	            #sdi_RunningTime := 0;
	            //Reset period caouter
	            #slr_PeriodMS := 0;

	        END_IF;
	    ELSE
	        // If FIFO is full set FIFO main and FIFO full errors.
	        #ss_Status.FIFOError := TRUE;
	        #ss_Status.FIFOStatus.FifoFull := TRUE;
	    END_IF;

	END_REGION

	REGION 5 - Status

	    // Parametrization collective error output.
	    #qx_Error :=
	    #ss_Status.FIFOError
	    OR #ss_Status.InvalidTimeInterval
	    OR #ss_Status.InvalidMessageArraySize;

	    // Parametrization collective warning output.
	    #qx_Warning := #ss_Status.FIFOWarning;

	END_REGION
END_FUNCTION_BLOCK

FUNCTION_BLOCK "FB_MFC_Sort_ParcelCounter"
{ S7_Optimized_Access := 'TRUE' }
VERSION : 0.1
// ATTRIBUTES
// AUTO_NUMBER = True
// BLOCK_NUMBER = 122
// END_ATTRIBUTES
   VAR_INPUT
      iui_LocationIdentifier { ExternalAccessible := 'False'; ExternalVisible := 'False'; ExternalWritable := 'False'} : UInt;   // SNCY finger identifier
      ix_Trigger { ExternalAccessible := 'False'; ExternalVisible := 'False'; ExternalWritable := 'False'} : Bool;   // A trigger that active message generation.
      ii_SourceNode { ExternalAccessible := 'False'; ExternalVisible := 'False'; ExternalWritable := 'False'} : Int;   // ID Source Node
      ii_DestinationNode { ExternalAccessible := 'False'; ExternalVisible := 'False'; ExternalWritable := 'False'} : Int;   // ID Destination Node
   END_VAR

   VAR_OUTPUT
      qx_Error { ExternalAccessible := 'False'; ExternalVisible := 'False'; ExternalWritable := 'False'} : Bool;   // TRUE when collective block error occurred
      qx_Warning { ExternalAccessible := 'False'; ExternalVisible := 'False'; ExternalWritable := 'False'} : Bool;   // TRUE when collective block warning occurred
   END_VAR

   VAR_IN_OUT
      iq_UDT_FifoHeader : "UDT_FifoHeader";   // FIFO header
      iqs_FifoData : Array[*] of "UDT_MessageV2";   // FIFO data buffer
      iqdi_MessageSequenceNumber { ExternalAccessible := 'False'; ExternalVisible := 'False'; ExternalWritable := 'False'} : Int;   // Message number
   END_VAR

   VAR
      s_UDT_MessageArray { ExternalAccessible := 'False'; ExternalVisible := 'False'; ExternalWritable := 'False'; S7_SetPoint := 'False'} : "UDT_MessageV2";   // Message array byte
      s_UDT_MessageHeader { ExternalAccessible := 'False'; ExternalVisible := 'False'; ExternalWritable := 'False'; S7_SetPoint := 'False'} : "UDT_MFCSortMessageHeader";   // Message header
      ss_MessageBody { ExternalAccessible := 'False'; ExternalVisible := 'False'; ExternalWritable := 'False'} : Struct   // Message body
         MsgID { ExternalAccessible := 'False'; ExternalVisible := 'False'; ExternalWritable := 'False'} : Word;   // Message ID
         MsgLength { ExternalAccessible := 'False'; ExternalVisible := 'False'; ExternalWritable := 'False'} : Word;   // Message length
         LocationIdentifier { ExternalAccessible := 'False'; ExternalVisible := 'False'; ExternalWritable := 'False'} : Word;   // Location Identifier
         Counts { ExternalAccessible := 'False'; ExternalVisible := 'False'; ExternalWritable := 'False'} : Word;   // Counts
         Eom { ExternalAccessible := 'False'; ExternalVisible := 'False'; ExternalWritable := 'False'} : Byte;   // End of message
      END_STRUCT;
      ss_Status { ExternalAccessible := 'False'; ExternalVisible := 'False'; ExternalWritable := 'False'} : Struct   // Status structure
         FIFOStatus { ExternalAccessible := 'False'; ExternalVisible := 'False'; ExternalWritable := 'False'} : "UDT_FifoStatus";
         FIFOError { ExternalAccessible := 'False'; ExternalVisible := 'False'; ExternalWritable := 'False'; S7_SetPoint := 'True'} : Bool;   //  FIFO error
         FIFOWarning { ExternalAccessible := 'False'; ExternalVisible := 'False'; ExternalWritable := 'False'; S7_SetPoint := 'True'} : Bool;   // FIFO warning
         InvalidMessageArraySize { ExternalAccessible := 'False'; ExternalVisible := 'False'; ExternalWritable := 'False'} : Bool;   // Message array is too short for message
         InvalidTimeInterval { ExternalAccessible := 'False'; ExternalVisible := 'False'; ExternalWritable := 'False'} : Bool;   // Heartbeat time interval lower than zero
      END_STRUCT;
      R_TRIG_SensorActive {InstructionName := 'R_TRIG'; LibVersion := '1.0'; ExternalAccessible := 'False'; ExternalVisible := 'False'; ExternalWritable := 'False'; S7_SetPoint := 'False'} : R_TRIG;   // Rising edge trigger from sensor
      sdi_SerializePosition { ExternalAccessible := 'False'; ExternalVisible := 'False'; ExternalWritable := 'False'} : DInt;   // Position in array where serialize finished writing data +1
      si_MaximumMessageLength { ExternalAccessible := 'False'; ExternalVisible := 'False'; ExternalWritable := 'False'} : Int;   // Maximum number of elements in message array
      si_SerializeStatus { ExternalAccessible := 'False'; ExternalVisible := 'False'; ExternalWritable := 'False'} : Int;   // Function serialize status
   END_VAR

   VAR CONSTANT
      ci_MessageLength : Word := 16#0008;   // 10#0008 = 16#0008 - Message length
      ci_Som : Byte := 16#FD;   // Start of message
      ci_Eom : Byte := 16#FE;   // End of message
      ci_MsgID : Word := 16#00CD;   // 10#0205 = 16#00CD - Message ID
      ci_MsgLength : Word := 16#0004;   // 10#0004 = 16#0004 - Message length
   END_VAR


BEGIN
	(*
	----------------------------------------------------------------------------------------
	|                                                                                      |
	|  Copyright  2023             FORTNA Europe BV                                        |
	|  All Rights Reserved         Netherlands                                             |
	|                                                                                      |
	----------------------------------------------------------------------------------------
	Version history:
	Date        | Version   | Author       | Remark
	----------------------------------------------------------------------------------------
	05/01/2023  | 1.0       | S. Nikodem   | Release TIA 17 | DHL Munich 2023
	13/03/2023  | 1.1       | S. Nieswiec  | Updated for new Baseline
	02/05/2024  | 4.2       | J.Majer      | Datatype conversions changed from automatic to explicit, to accomodate IEC 61131-3 standard

	*)

	REGION 1 – FIFO header status update

	    // Mode 'S' - FIFO register status update.
	    "FC_Fifo"(ic_Mode := 'S',
	              qUDT_Status => #ss_Status.FIFOStatus,
	              qx_Error => #ss_Status.FIFOError,
	              qx_Warning => #ss_Status.FIFOWarning,
	              iqv_Data := #s_UDT_MessageArray,
	              iqUDT_FifoHeader := #iq_UDT_FifoHeader,
	              iqv_DataBuffer := #iqs_FifoData);

	END_REGION

	REGION 2 – Data preparation

	    #R_TRIG_SensorActive(CLK := #ix_Trigger);

	END_REGION

	REGION 3 – Message array size validation

	    // Get size of the array.
	    #si_MaximumMessageLength := "FC_GetNrOfArrayEl"(#s_UDT_MessageArray.Bytes);

	    // Message array size validation.
	    #ss_Status.InvalidMessageArraySize := WORD_TO_INT(#ci_MessageLength) > #si_MaximumMessageLength;

	END_REGION


	REGION 4 – Message preparation

	    // FIFO full check.
	    IF NOT #iq_UDT_FifoHeader.Status.Full
	    THEN
	        // Errors and send pulse check.
	        IF NOT #ss_Status.FIFOError
	            AND NOT #ss_Status.InvalidMessageArraySize
	            AND #R_TRIG_SensorActive.Q
	        THEN

	            REGION 4.1 – Header preparation

	                // Check sequence number. If it is equal or greater than 255 reset it to 1.
	                IF #iqdi_MessageSequenceNumber <= 255
	                THEN
	                    #iqdi_MessageSequenceNumber += 1;
	                ELSE
	                    #iqdi_MessageSequenceNumber := 1;
	                END_IF;

	                // Write parts of the header into structure.
	                #s_UDT_MessageHeader.SOM := #ci_Som;
	                #s_UDT_MessageHeader.SourceNode := INT_TO_BYTE(#ii_SourceNode);
	                #s_UDT_MessageHeader.DestinationNode := INT_TO_BYTE(#ii_DestinationNode);
	                #s_UDT_MessageHeader.SeqNumber := INT_TO_BYTE(#iqdi_MessageSequenceNumber);
	                #s_UDT_MessageHeader.DataLength := #ci_MessageLength;
	                #s_UDT_MessageHeader.NumMsg := 1;

	                // Write parts of the body into structure.
	                #ss_MessageBody.MsgID := #ci_MsgID;
	                #ss_MessageBody.MsgLength := #ci_MsgLength;
	                #ss_MessageBody.LocationIdentifier := DINT_TO_WORD(#iui_LocationIdentifier);
	                #ss_MessageBody.Counts := 1;
	                #ss_MessageBody.Eom := #ci_Eom;

	            END_REGION

	            REGION 4.2 – Convert message into array of bytes

	                // Initialize the header serialize position and convert header structure into array of bytes.
	                #sdi_SerializePosition := 0;
	                #si_SerializeStatus := Serialize(SRC_VARIABLE := #s_UDT_MessageHeader,
	                                                 DEST_ARRAY => #s_UDT_MessageArray.Bytes,
	                                                 POS := #sdi_SerializePosition);

	                // Initialize the body serialize position and convert header structure into array of bytes
	                #si_SerializeStatus := Serialize(SRC_VARIABLE := #ss_MessageBody,
	                                                 DEST_ARRAY => #s_UDT_MessageArray.Bytes,
	                                                 POS := #sdi_SerializePosition);

	            END_REGION

	            REGION 4.3 – Write message into the FIFO buffer

	                // Mode 'W' - Write FIFO record.
	                "FC_Fifo"(ic_Mode := 'W',
	                          qUDT_Status => #ss_Status.FIFOStatus,
	                          qx_Error => #ss_Status.FIFOError,
	                          qx_Warning => #ss_Status.FIFOWarning,
	                          iqv_Data := #s_UDT_MessageArray,
	                          iqUDT_FifoHeader := #iq_UDT_FifoHeader,
	                          iqv_DataBuffer := #iqs_FifoData);

	            END_REGION

	        END_IF;
	    ELSE
	        // If FIFO is full set FIFO main and FIFO full errors.
	        #ss_Status.FIFOError := TRUE;
	        #ss_Status.FIFOStatus.FifoFull := TRUE;
	    END_IF;

	END_REGION

	REGION 5 - Status

	    // Parametrization collective error output.
	    #qx_Error :=
	    #ss_Status.FIFOError
	    OR #ss_Status.InvalidTimeInterval
	    OR #ss_Status.InvalidMessageArraySize;

	    // Parametrization collective warning output.
	    #qx_Warning := #ss_Status.FIFOWarning;

	END_REGION
END_FUNCTION_BLOCK

FUNCTION_BLOCK "FB_MFC_Sort_ScanReset"
{ S7_Optimized_Access := 'TRUE' }
VERSION : 0.1
// ATTRIBUTES
// AUTO_NUMBER = True
// BLOCK_NUMBER = 123
// END_ATTRIBUTES
   VAR_INPUT
      is_ObjectID { ExternalAccessible := 'False'; ExternalVisible := 'False'; ExternalWritable := 'False'} : String[10];   // Parcel identifier
      ii_SourceNode { ExternalAccessible := 'False'; ExternalVisible := 'False'; ExternalWritable := 'False'} : Int;   // ID Source Node
      ii_DestinationNode { ExternalAccessible := 'False'; ExternalVisible := 'False'; ExternalWritable := 'False'} : Int;   // ID Destination Node
   END_VAR

   VAR_OUTPUT
      qx_Error { ExternalAccessible := 'False'; ExternalVisible := 'False'; ExternalWritable := 'False'} : Bool;   // TRUE when collective block error occurred
      qx_Warning { ExternalAccessible := 'False'; ExternalVisible := 'False'; ExternalWritable := 'False'} : Bool;   // TRUE when collective block warning occurred
   END_VAR

   VAR_IN_OUT
      iq_UDT_FifoHeader : "UDT_FifoHeader";   // FIFO header
      iqs_FifoData : Array[*] of "UDT_MessageV2";   // FIFO data buffer
      iqdi_MessageSequenceNumber { ExternalAccessible := 'False'; ExternalVisible := 'False'; ExternalWritable := 'False'} : Int;   // Message number
   END_VAR

   VAR
      ss_FB_HeartbeatPulse { ExternalAccessible := 'False'; ExternalVisible := 'False'; ExternalWritable := 'False'; S7_SetPoint := 'False'} : "FB_Pulse";   // Heartbeat send pulse generator
      s_UDT_MessageArray { ExternalAccessible := 'False'; ExternalVisible := 'False'; ExternalWritable := 'False'; S7_SetPoint := 'False'} : "UDT_MessageV2";   // Message array byte
      s_UDT_MessageHeader { ExternalAccessible := 'False'; ExternalVisible := 'False'; ExternalWritable := 'False'; S7_SetPoint := 'False'} : "UDT_MFCSortMessageHeader";   // Message header
      ss_MessageBody { ExternalAccessible := 'False'; ExternalVisible := 'False'; ExternalWritable := 'False'} : Struct   // Message body
         MsgID { ExternalAccessible := 'False'; ExternalVisible := 'False'; ExternalWritable := 'False'} : Word;   // Message ID
         MsgLength { ExternalAccessible := 'False'; ExternalVisible := 'False'; ExternalWritable := 'False'} : Word;   // Message length
         ObjectID { ExternalAccessible := 'False'; ExternalVisible := 'False'; ExternalWritable := 'False'} : DWord;   // Parcel identifier
         Eom { ExternalAccessible := 'False'; ExternalVisible := 'False'; ExternalWritable := 'False'} : Byte;   // End of message
      END_STRUCT;
      ss_Status { ExternalAccessible := 'False'; ExternalVisible := 'False'; ExternalWritable := 'False'} : Struct   // Status structure
         FIFOStatus { ExternalAccessible := 'False'; ExternalVisible := 'False'; ExternalWritable := 'False'} : "UDT_FifoStatus";
         FIFOError { ExternalAccessible := 'False'; ExternalVisible := 'False'; ExternalWritable := 'False'; S7_SetPoint := 'True'} : Bool;   //  FIFO error
         FIFOWarning { ExternalAccessible := 'False'; ExternalVisible := 'False'; ExternalWritable := 'False'; S7_SetPoint := 'True'} : Bool;   // FIFO warning
         InvalidMessageArraySize { ExternalAccessible := 'False'; ExternalVisible := 'False'; ExternalWritable := 'False'} : Bool;   // Message array is too short for message
         InvalidTimeInterval { ExternalAccessible := 'False'; ExternalVisible := 'False'; ExternalWritable := 'False'} : Bool;   // Heartbeat time interval lower than zero
      END_STRUCT;
      sdi_SerializePosition { ExternalAccessible := 'False'; ExternalVisible := 'False'; ExternalWritable := 'False'} : DInt;   // Position in array where serialize finished writing data +1
      si_MaximumMessageLength { ExternalAccessible := 'False'; ExternalVisible := 'False'; ExternalWritable := 'False'} : Int;   // Maximum number of elements in message array
      si_SerializeStatus { ExternalAccessible := 'False'; ExternalVisible := 'False'; ExternalWritable := 'False'} : Int;   // Function serialize status
      ss_Old_Object_ID { ExternalAccessible := 'False'; ExternalVisible := 'False'; ExternalWritable := 'False'} : String[10];   // Value from previous PLC cycle
      sx_NewData { ExternalAccessible := 'False'; ExternalVisible := 'False'; ExternalWritable := 'False'} : Bool;   // True - send a message to the MFC
      sa_EmptyObjectID { ExternalAccessible := 'False'; ExternalVisible := 'False'; ExternalWritable := 'False'} : Array[1..10] of Byte;   // Parcel identifier
   END_VAR

   VAR_TEMP
      tudi_Temp : UDInt;
   END_VAR

   VAR CONSTANT
      ci_MessageLength : Word := 16#0006;   // 10#0006 = 16#0006 - Message length
      ci_Som : Byte := 16#FD;   // Start of message
      ci_Eom : Byte := 16#FE;   // End of message
      ci_MsgID : Word := 16#00CA;   // 10#0202 = 16#00CA - Message ID
      ci_MsgLength : Word := 16#0002;   // 10#0002 = 16#0002 - Message length
   END_VAR


BEGIN
	(*
	----------------------------------------------------------------------------------------
	|                                                                                      |
	|  Copyright  2023             FORTNA Europe BV                                        |
	|  All Rights Reserved         Netherlands                                             |
	|                                                                                      |
	----------------------------------------------------------------------------------------
	Version history:
	Date        | Version   | Author       | Remark
	----------------------------------------------------------------------------------------
	05/01/2023  | 1.0       | S. Nikodem   | Release TIA 17 | DHL Munich 2023
	13/03/2023  | 1.1       | S. Nieswiec  | Updated for new Baseline
	02/05/2024  | 1.2       | J.Majer      | Datatype conversions changed from automatic to explicit, to accomodate IEC 61131-3 standard

	*)

	REGION 1 – FIFO header status update

	    // Mode 'S' - FIFO register status update.
	    "FC_Fifo"(ic_Mode := 'S',
	              qUDT_Status => #ss_Status.FIFOStatus,
	              qx_Error => #ss_Status.FIFOError,
	              qx_Warning => #ss_Status.FIFOWarning,
	              iqv_Data := #s_UDT_MessageArray,
	              iqUDT_FifoHeader := #iq_UDT_FifoHeader,
	              iqv_DataBuffer := #iqs_FifoData);

	END_REGION

	REGION 2 – Data preparation

